       IF NOT #Positionen[20].Sperre AND NOT #Vorzug THEN
           "FC_FW_Auftrag_Befehl"(inQuelle := #tmpQuelle,
                                  inZiel := 20,
                                  Befehl_ok => #Befehl_ok,
                                  outQuelle => #Quelle,
                                  outZiel => #Ziel);

           #nextStep := NOT #Befehl_ok;
       ELSIF NOT #Positionen[24].Sperre THEN
           "FC_FW_Auftrag_Befehl"(inQuelle := #tmpQuelle,
                                  inZiel := 24,
                                  Befehl_ok => #Befehl_ok,
                                  outQuelle => #Quelle,
                                  outZiel => #Ziel);

           #nextStep := NOT #Befehl_ok;
       ELSE
           #nextStep := TRUE;
       END_IF;
       RETURN;
   END_IF;

   //
   #nextStep := TRUE;
END_REGION
END_FUNCTION

FUNCTION "FC_FW_Auftrag_Step1_NB" : Void   // FC181, LAD
TITLE = Schritt CM01/CMD02 -> CM03
{ S7_Optimized_Access := 'TRUE' }
// Ältesten Warenträger in CM01/CM02 suchen und nach CM03 transportieren
// stored: AutoNumber false, SetENOAutomatically false
   VAR_INPUT
      Frg_Schritt : Bool;
   END_VAR
   VAR_OUTPUT
      nextStep : Bool;
      startStep : Bool;
      parkStep : Bool;
   END_VAR
   VAR_IN_OUT
      Quelle : Int;
      Ziel : Int;
      Positionen : Array[1..30] of "UDT_Auftrag_Pos";
   END_VAR
   VAR_TEMP
      Sperre_Kurz_li : Bool;
      Sperre_Kurz_re : Bool;
      Sperre_Lang : Bool;
      Vorzug : Bool;
      Befehl_ok : Bool;
      tmpQuelle : Int;
      Oldest : Real;
   END_VAR
BEGIN

REGION Network 1 (SCL): Initialisieren
   IF (#Quelle <> 0) AND (#Ziel <> 0) THEN
       #nextStep := #Positionen[#Quelle].Sperre;
       #startStep := NOT #nextStep;
       #Quelle := 0;
       #Ziel := 0;
       RETURN;
   END_IF;

   #Quelle := 0;
   #Ziel := 0;
   #nextStep := FALSE;
   #startStep := FALSE;

   IF NOT #Frg_Schritt THEN
       #nextStep := TRUE;
       RETURN;
   END_IF;
END_REGION

REGION Network 2 (SCL): Positionen sperren
   //Groß links nicht möglich
   #Positionen[3].CheckSperre := #Positionen[9].Sperre;
   #Positionen[15].CheckSperre := #Positionen[9].Sperre;

   //Groß rechts nicht möglich
   #Positionen[4].CheckSperre := #Positionen[10].Sperre;
   #Positionen[16].CheckSperre := #Positionen[10].Sperre;

   //kein Platz für Kurz links in CM03
   #Sperre_Kurz_li := #Positionen[7].Sperre AND #Positionen[11].Sperre;

   //kein Platz für Kurz rechts in CM03
   #Sperre_Kurz_re := #Positionen[8].Sperre AND #Positionen[12].Sperre;

   //kein Platz für Lang in CM03
   #Sperre_Lang := (#Positionen[7].Sperre OR #Positionen[8].Sperre) AND (#Positionen[11].Sperre OR #Positionen[12].Sperre);

   //Lang in P1 oder
   //kein Platz auf rechter Seite
   //-> P2 sperren
   #Positionen[2].CheckSperre := #Sperre_Kurz_re OR (#Positionen[1].Wt_Typ = "WT_Typ_LS");

   //Lang in P1 und kein Platz für Lang oder
   //kein Platz auf linker Seite
   //-> P1 sperren
   #Positionen[1].CheckSperre := #Sperre_Kurz_li OR ((#Positionen[1].Wt_Typ = "WT_Typ_LS") AND #Sperre_Lang);

   //Lang in P5 oder
   //kein Platz auf rechter Seite
   //-> P6 sperren
   #Positionen[6].CheckSperre := #Sperre_Kurz_re OR (#Positionen[5].Wt_Typ = "WT_Typ_LS");

   //Lang in P5 und kein Platz für Lang oder
   //kein Platz auf linker Seite
   //-> P5 sperren
   #Positionen[5].CheckSperre := #Sperre_Kurz_li OR ((#Positionen[5].Wt_Typ = "WT_Typ_LS") AND #Sperre_Lang);

   //Lang in P13 oder
   //kein Platz auf rechter Seite
   //-> P14 sperren
   #Positionen[14].CheckSperre := #Sperre_Kurz_re OR (#Positionen[13].Wt_Typ = "WT_Typ_LS");

   //Lang in P13 und kein Platz für Lang oder
   //kein Platz auf linker Seite
   //-> P13 sperren
   #Positionen[13].CheckSperre := #Sperre_Kurz_li OR ((#Positionen[13].Wt_Typ = "WT_Typ_LS") AND #Sperre_Lang);

   //Lang in P17 oder
   //kein Platz auf rechter Seite
   //-> P18 sperren
   #Positionen[18].CheckSperre := #Sperre_Kurz_re OR (#Positionen[17].Wt_Typ = "WT_Typ_LS");

   //Lang in P17 und kein Platz für Lang oder
   //kein Platz auf linker Seite
   //-> P17 sperren
   #Positionen[17].CheckSperre := #Sperre_Kurz_li OR ((#Positionen[17].Wt_Typ = "WT_Typ_LS") AND #Sperre_Lang);
END_REGION

REGION Network 3 (SCL): Ältesten WT suchen
   //
   #Oldest := 0;
   #tmpQuelle := 0;

   //CM01
   "FC_FW_Auftrag_Suche"(Pos1 := 1,
                         Pos2 := 6,
                         Positionen := #Positionen,
                         Quelle := #tmpQuelle,
                         Oldest := #Oldest);

   //CM02
   "FC_FW_Auftrag_Suche"(Pos1 := 13,
                         Pos2 := 18,
                         Positionen := #Positionen,
                         Quelle := #tmpQuelle,
                         Oldest := #Oldest);
END_REGION

REGION Network 4 (SCL): Auswertung
   IF #tmpQuelle = 0 THEN
       //kein WT
       #nextStep := TRUE;
       RETURN;
   END_IF;

   IF ("DI_FW_1".ZST.POSITION_li <= 6) AND (#tmpQuelle <= 6) THEN
       //schieben wenn über Quelle CM01
       "FC_FW_Auftrag_Befehl"(inQuelle := 7,
                              inZiel := 0,
                              Befehl_ok => #Befehl_ok,
                              outQuelle => #Quelle,
                              outZiel => #Ziel);

       #nextStep := NOT #Befehl_ok;
       RETURN;
   END_IF;

   IF ("DI_FW_1".ZST.POSITION_li >= 13) AND ("DI_FW_1".ZST.POSITION_li <= 18) AND (#tmpQuelle >= 13) THEN
       //schieben wenn über Quelle CM02
       "FC_FW_Auftrag_Befehl"(inQuelle := 11,
                              inZiel := 0,
                              Befehl_ok => #Befehl_ok,
                              outQuelle => #Quelle,
                              outZiel => #Ziel);

       #nextStep := NOT #Befehl_ok;
       RETURN;
   END_IF;

   IF NOT #Positionen[#tmpQuelle].Fertig THEN
       #parkStep := TRUE;
       RETURN;
   END_IF;

   IF (#tmpQuelle = 3) OR (#tmpQuelle = 15) THEN
       //Gross links
       IF NOT #Positionen[9].Sperre THEN
           "FC_FW_Auftrag_Befehl"(inQuelle := #tmpQuelle,
                                  inZiel := 9,
                                  Befehl_ok => #Befehl_ok,
                                  outQuelle => #Quelle,
                                  outZiel => #Ziel);

           #nextStep := NOT #Befehl_ok;
       ELSE
           #nextStep := TRUE;
       END_IF;
       RETURN;
   END_IF;

   IF (#tmpQuelle = 4) OR (#tmpQuelle = 16) THEN
       //Gross rechts
       IF NOT #Positionen[10].Sperre THEN
           "FC_FW_Auftrag_Befehl"(inQuelle := #tmpQuelle,
                                  inZiel := 10,
                                  Befehl_ok => #Befehl_ok,
                                  outQuelle => #Quelle,
                                  outZiel => #Ziel);

           #nextStep := NOT #Befehl_ok;
       ELSE
           #nextStep := TRUE;
       END_IF;
       RETURN;
   END_IF;

   IF (#Positionen[#tmpQuelle].Wt_Typ = "WT_Typ_LS") AND ((#tmpQuelle = 1) OR (#tmpQuelle = 5) OR (#tmpQuelle = 13) OR (#tmpQuelle = 17)) THEN
       //Lang
       IF NOT #Positionen[7].Sperre AND NOT #Positionen[8].Sperre THEN
           "FC_FW_Auftrag_Befehl"(inQuelle := #tmpQuelle,
                                  inZiel := 7,
                                  Befehl_ok => #Befehl_ok,
                                  outQuelle => #Quelle,
                                  outZiel => #Ziel);

           #nextStep := NOT #Befehl_ok;
       ELSIF NOT #Positionen[11].Sperre AND NOT #Positionen[12].Sperre THEN
           "FC_FW_Auftrag_Befehl"(inQuelle := #tmpQuelle,
                                  inZiel := 11,
                                  Befehl_ok => #Befehl_ok,
                                  outQuelle => #Quelle,
                                  outZiel => #Ziel);

           #nextStep := NOT #Befehl_ok;
       ELSE
           #nextStep := TRUE;
       END_IF;
       RETURN;
   END_IF;

   IF (#tmpQuelle = 1) OR (#tmpQuelle = 5) OR (#tmpQuelle = 13) OR (#tmpQuelle = 17) THEN
       //Kurz links
       #Vorzug := NOT #Positionen[7].Sperre AND NOT #Positionen[8].Sperre AND NOT #Positionen[11].Sperre AND #Positionen[12].Sperre;

       IF NOT #Positionen[7].Sperre AND NOT #Vorzug THEN
           "FC_FW_Auftrag_Befehl"(inQuelle := #tmpQuelle,
                                  inZiel := 7,
                                  Befehl_ok => #Befehl_ok,
                                  outQuelle => #Quelle,
                                  outZiel => #Ziel);

           #nextStep := NOT #Befehl_ok;
       ELSIF NOT #Positionen[11].Sperre THEN
           "FC_FW_Auftrag_Befehl"(inQuelle := #tmpQuelle,
                                  inZiel := 11,
                                  Befehl_ok => #Befehl_ok,
                                  outQuelle => #Quelle,
                                  outZiel => #Ziel);

           #nextStep := NOT #Befehl_ok;
       ELSE
           #nextStep := TRUE;
       END_IF;
       RETURN;
   END_IF;

   IF (#tmpQuelle = 2) OR (#tmpQuelle = 6) OR (#tmpQuelle = 14) OR (#tmpQuelle = 18) THEN
       //Kurz rechts
       #Vorzug := NOT #Positionen[7].Sperre AND NOT #Positionen[8].Sperre AND #Positionen[11].Sperre AND NOT #Positionen[12].Sperre;

       IF NOT #Positionen[8].Sperre AND NOT #Vorzug THEN
           "FC_FW_Auftrag_Befehl"(inQuelle := #tmpQuelle,
                                  inZiel := 8,
                                  Befehl_ok => #Befehl_ok,
                                  outQuelle => #Quelle,
                                  outZiel => #Ziel);

           #nextStep := NOT #Befehl_ok;
       ELSIF NOT #Positionen[12].Sperre THEN
           "FC_FW_Auftrag_Befehl"(inQuelle := #tmpQuelle,
                                  inZiel := 12,
                                  Befehl_ok => #Befehl_ok,
                                  outQuelle => #Quelle,
                                  outZiel => #Ziel);

           #nextStep := NOT #Befehl_ok;
       ELSE
           #nextStep := TRUE;
       END_IF;
       RETURN;
   END_IF;

   //?
   #nextStep := TRUE;
END_REGION
END_FUNCTION

FUNCTION "FC_FW_Auftrag_Step2_KB" : Void   // FC1082, LAD
TITLE = Schritt CM03/CM04 -> CM01/CM02
{ S7_Optimized_Access := 'TRUE' }
// Ältesten Warenträger in CM03/CM04 suchen und nach CM01/CM02 transportieren
// stored: AutoNumber false, SetENOAutomatically false
   VAR_INPUT
      Frg_Schritt : Bool;
   END_VAR
   VAR_OUTPUT
      nextStep : Bool;
      startStep : Bool;
      parkStep : Bool;
   END_VAR
   VAR_IN_OUT
      Quelle : Int;
      Ziel : Int;
      Positionen : Array[1..30] of "UDT_Auftrag_Pos";
   END_VAR
   VAR_TEMP
      Sperre_Kurz_li_CM01 : Bool;
      Sperre_Kurz_re_CM01 : Bool;
      Sperre_Lang_CM01 : Bool;
      Sperre_Kurz_li_CM02 : Bool;
      Sperre_Kurz_re_CM02 : Bool;
      Sperre_Lang_CM02 : Bool;
      Vorzug : Bool;
      Vorzug1 : Bool;
      Vorzug2 : Bool;
      Befehl_ok : Bool;
      tmpQuelle : Int;
      Oldest : Real;
   END_VAR
   VAR CONSTANT
      Wt_Cmd_AetzenCM01 : Int := 1;
      Wt_Cmd_AetzenCM02 : Int := 13;
   END_VAR
BEGIN

REGION Network 1 (SCL)
   IF (#Quelle <> 0) AND (#Ziel <> 0) THEN
       #nextStep := #Positionen[#Quelle].Sperre;
       #startStep := NOT #nextStep;
       #Quelle := 0;
       #Ziel := 0;
       RETURN;
   END_IF;

   #Quelle := 0;
   #Ziel := 0;
   #nextStep := FALSE;
   #startStep := FALSE;

   IF NOT #Frg_Schritt THEN
       #nextStep := TRUE;
       RETURN;
   END_IF;
END_REGION

REGION Network 2 (SCL): Positionen sperren
   // GO nur "161"
   //Groß links nicht möglich
   #Positionen[9].CheckSperre := (#Positionen[3].Sperre ) OR (#Positionen[9].Wt_Cmd <> #Wt_Cmd_AetzenCM01);

   //Groß rechts nicht möglich
   #Positionen[10].CheckSperre := (#Positionen[4].Sperre AND #Positionen[16].Sperre) OR (#Positionen[10].Wt_Cmd <> #Wt_Cmd_AetzenCM01);

   //kein Platz für Kurz links in CM01
   #Sperre_Kurz_li_CM01 := #Positionen[1].Sperre AND #Positionen[5].Sperre;

   //kein Platz für Kurz links in CM02
   #Sperre_Kurz_li_CM02 := #Positionen[13].Sperre AND #Positionen[17].Sperre;

   //kein Platz für Kurz rechts in CM01
   #Sperre_Kurz_re_CM01 := #Positionen[2].Sperre AND #Positionen[6].Sperre;

   //kein Platz für Kurz rechts in CM02
   #Sperre_Kurz_re_CM02 := #Positionen[14].Sperre AND #Positionen[18].Sperre;

   //kein Platz für Lang in CM01
   #Sperre_Lang_CM01 := (#Positionen[1].Sperre OR #Positionen[2].Sperre) AND (#Positionen[5].Sperre OR #Positionen[6].Sperre);

   //kein Platz für Lang in CM02
   #Sperre_Lang_CM02:= (#Positionen[13].Sperre OR #Positionen[14].Sperre) AND (#Positionen[17].Sperre OR #Positionen[18].Sperre);

   //Lang in P7 oder
   //kein Platz auf rechter Seite
   //-> P8 sperren
   #Positionen[8].CheckSperre := #Sperre_Kurz_re_CM01 OR (#Positionen[7].Wt_Typ = "WT_Typ_LS") OR (#Positionen[8].Wt_Cmd <> #Wt_Cmd_AetzenCM01);

   //Lang in P7 und kein Platz für Lang oder
   //kein Platz auf linker Seite
   //-> P7 sperren
   #Positionen[7].CheckSperre := #Sperre_Kurz_li_CM01 OR ((#Positionen[7].Wt_Typ = "WT_Typ_LS") AND #Sperre_Lang_CM01) OR (#Positionen[7].Wt_Cmd <> #Wt_Cmd_AetzenCM01);

   //Lang in P7 oder
   //kein Platz auf rechter Seite
   //-> P12 sperren
   #Positionen[12].CheckSperre := #Sperre_Kurz_re_CM01 OR (#Positionen[11].Wt_Typ = "WT_Typ_LS") OR (#Positionen[12].Wt_Cmd <> #Wt_Cmd_AetzenCM01);

   //Lang in P11 und kein Platz für Lang oder
   //kein Platz auf linker Seite
   //-> P11 sperren
   #Positionen[11].CheckSperre := #Sperre_Kurz_li_CM01 OR ((#Positionen[11].Wt_Typ = "WT_Typ_LS") AND #Sperre_Lang_CM01) OR (#Positionen[11].Wt_Cmd <> #Wt_Cmd_AetzenCM01);

   //Lang in P19 oder
   //kein Platz auf rechter Seite
   //-> P20 sperren
   #Positionen[20].CheckSperre := #Sperre_Kurz_re_CM02 OR (#Positionen[19].Wt_Typ = "WT_Typ_LS") OR (#Positionen[20].Wt_Cmd <> #Wt_Cmd_AetzenCM02);

   //Lang in P19 und kein Platz für Lang oder
   //kein Platz auf linker Seite
   //-> P19 sperren
   #Positionen[19].CheckSperre := #Sperre_Kurz_li_CM02 OR ((#Positionen[19].Wt_Typ = "WT_Typ_LS") AND #Sperre_Lang_CM02) OR (#Positionen[19].Wt_Cmd <> #Wt_Cmd_AetzenCM02);

   //Lang in P23 oder
   //kein Platz auf rechter Seite
   //-> P24 sperren
   #Positionen[24].CheckSperre := #Sperre_Kurz_re_CM02 OR (#Positionen[23].Wt_Typ = "WT_Typ_LS") OR (#Positionen[24].Wt_Cmd <> #Wt_Cmd_AetzenCM02);

   //Lang in P23 und kein Platz für Lang oder
   //kein Platz auf linker Seite
   //-> P23 sperren
   #Positionen[23].CheckSperre := #Sperre_Kurz_li_CM02 OR ((#Positionen[23].Wt_Typ = "WT_Typ_LS") AND #Sperre_Lang_CM02) OR (#Positionen[23].Wt_Cmd <> #Wt_Cmd_AetzenCM02);
END_REGION

REGION Network 3 (SCL): Ältesten WT suchen
   //
   #Oldest := 0;
   #tmpQuelle := 0;

   //CM03
   "FC_FW_Auftrag_Suche"(Pos1 := 7,
                         Pos2 := 12,
                         Positionen := #Positionen,
                         Quelle := #tmpQuelle,
                         Oldest := #Oldest);

   //CM04
   "FC_FW_Auftrag_Suche"(Pos1 := 19,
                         Pos2 := 24,
                         Positionen := #Positionen,
                         Quelle := #tmpQuelle,
                         Oldest := #Oldest);
END_REGION

REGION Network 4 (SCL): Auswertung
   IF #tmpQuelle = 0 THEN
       //kein WT
       #nextStep := TRUE;
       RETURN;
   END_IF;

   IF NOT #Positionen[#tmpQuelle].Fertig THEN
       #parkStep := TRUE;
       RETURN;
   END_IF;

   IF (#tmpQuelle = 9) THEN
       //Gross links nur "161"
       IF NOT #Positionen[3].Sperre THEN
           "FC_FW_Auftrag_Befehl"(inQuelle := #tmpQuelle,
                                  inZiel := 3,
                                  Befehl_ok => #Befehl_ok,
                                  outQuelle => #Quelle,
                                  outZiel => #Ziel);

           #nextStep := NOT #Befehl_ok;
       ELSE
           #nextStep := TRUE;
       END_IF;
       RETURN;
   END_IF;

   IF (#tmpQuelle = 10) THEN
       //Gross rechts nur "161"
       IF NOT #Positionen[4].Sperre THEN
           "FC_FW_Auftrag_Befehl"(inQuelle := #tmpQuelle,
                                  inZiel := 4,
                                  Befehl_ok => #Befehl_ok,
                                  outQuelle => #Quelle,
                                  outZiel => #Ziel);

           #nextStep := NOT #Befehl_ok;
       ELSE
           #nextStep := TRUE;
       END_IF;
       RETURN;
   END_IF;

   IF (#Positionen[#tmpQuelle].Wt_Typ = "WT_Typ_LS") AND ((#tmpQuelle = 7) OR (#tmpQuelle = 11)) THEN
       //Lang "161"
       IF NOT #Positionen[5].Sperre AND NOT #Positionen[6].Sperre THEN
           "FC_FW_Auftrag_Befehl"(inQuelle := #tmpQuelle,
                                  inZiel := 5,
                                  Befehl_ok => #Befehl_ok,
                                  outQuelle => #Quelle,
                                  outZiel => #Ziel);

           #nextStep := NOT #Befehl_ok;
       ELSIF NOT #Positionen[1].Sperre AND NOT #Positionen[2].Sperre THEN
           "FC_FW_Auftrag_Befehl"(inQuelle := #tmpQuelle,
                                  inZiel := 1,
                                  Befehl_ok => #Befehl_ok,
                                  outQuelle => #Quelle,
                                  outZiel => #Ziel);

           #nextStep := NOT #Befehl_ok;
       ELSE
           #nextStep := TRUE;
       END_IF;
       RETURN;
   END_IF;

   IF (#Positionen[#tmpQuelle].Wt_Typ = "WT_Typ_LS") AND ((#tmpQuelle = 19) OR (#tmpQuelle = 23)) THEN
       //Lang "151"
       IF NOT #Positionen[17].Sperre AND NOT #Positionen[18].Sperre THEN
           "FC_FW_Auftrag_Befehl"(inQuelle := #tmpQuelle,
                                  inZiel := 17,
                                  Befehl_ok => #Befehl_ok,
                                  outQuelle => #Quelle,
                                  outZiel => #Ziel);

           #nextStep := NOT #Befehl_ok;
       ELSIF NOT #Positionen[13].Sperre AND NOT #Positionen[14].Sperre THEN
           "FC_FW_Auftrag_Befehl"(inQuelle := #tmpQuelle,
                                  inZiel := 13,
                                  Befehl_ok => #Befehl_ok,
                                  outQuelle => #Quelle,
                                  outZiel => #Ziel);

           #nextStep := NOT #Befehl_ok;
       ELSE
           #nextStep := TRUE;
       END_IF;
       RETURN;
   END_IF;

   IF (#tmpQuelle = 7) OR (#tmpQuelle = 11) THEN
       //Kurz links "161"
       #Vorzug1 := NOT #Positionen[1].Sperre AND #Positionen[2].Sperre;
       #Vorzug2 := NOT #Positionen[5].Sperre AND #Positionen[6].Sperre;

       #Vorzug := NOT #Vorzug2 AND #Vorzug1;
       IF NOT #Positionen[5].Sperre AND NOT #Vorzug THEN
           "FC_FW_Auftrag_Befehl"(inQuelle := #tmpQuelle,
                                  inZiel := 5,
                                  Befehl_ok => #Befehl_ok,
                                  outQuelle => #Quelle,
                                  outZiel => #Ziel);

           #nextStep := NOT #Befehl_ok;
           RETURN;
       END_IF;

       #Vorzug := NOT #Vorzug1 AND #Vorzug1;
       IF NOT #Positionen[1].Sperre AND NOT #Vorzug THEN
           "FC_FW_Auftrag_Befehl"(inQuelle := #tmpQuelle,
                                  inZiel := 1,
                                  Befehl_ok => #Befehl_ok,
                                  outQuelle => #Quelle,
                                  outZiel => #Ziel);

           #nextStep := NOT #Befehl_ok;
           RETURN;
       END_IF;

       #nextStep := TRUE;
       RETURN;
   END_IF;

   IF (#tmpQuelle = 8) OR (#tmpQuelle = 12) THEN
       //Kurz rechts "161"
       #Vorzug1 := NOT #Positionen[2].Sperre AND #Positionen[1].Sperre;
       #Vorzug2 := NOT #Positionen[6].Sperre AND #Positionen[5].Sperre;

       #Vorzug := NOT #Vorzug2 AND #Vorzug1;
       IF NOT #Positionen[6].Sperre AND NOT #Vorzug THEN
           "FC_FW_Auftrag_Befehl"(inQuelle := #tmpQuelle,
                                  inZiel := 6,
                                  Befehl_ok => #Befehl_ok,
                                  outQuelle => #Quelle,
                                  outZiel => #Ziel);

           #nextStep := NOT #Befehl_ok;
           RETURN;
       END_IF;


       #Vorzug := NOT #Vorzug1 AND #Vorzug2;
       IF NOT #Positionen[2].Sperre AND NOT #Vorzug THEN
           "FC_FW_Auftrag_Befehl"(inQuelle := #tmpQuelle,
                                  inZiel := 2,
                                  Befehl_ok => #Befehl_ok,
                                  outQuelle => #Quelle,
                                  outZiel => #Ziel);

           #nextStep := NOT #Befehl_ok;
           RETURN;
       END_IF;

       #nextStep := TRUE;
       RETURN;
   END_IF;

   IF (#tmpQuelle = 19) OR (#tmpQuelle = 23) THEN
       //Kurz links "151"
       #Vorzug1 := NOT #Positionen[13].Sperre AND #Positionen[14].Sperre;
       #Vorzug2 := NOT #Positionen[17].Sperre AND #Positionen[18].Sperre;

       #Vorzug := NOT #Vorzug2 AND #Vorzug1;
       IF NOT #Positionen[17].Sperre AND NOT #Vorzug THEN
           "FC_FW_Auftrag_Befehl"(inQuelle := #tmpQuelle,
                                  inZiel := 17,
                                  Befehl_ok => #Befehl_ok,
                                  outQuelle => #Quelle,
                                  outZiel => #Ziel);

           #nextStep := NOT #Befehl_ok;
           RETURN;
       END_IF;

       #Vorzug := NOT #Vorzug1 AND #Vorzug1;
       IF NOT #Positionen[13].Sperre AND NOT #Vorzug THEN
           "FC_FW_Auftrag_Befehl"(inQuelle := #tmpQuelle,
                                  inZiel := 13,
                                  Befehl_ok => #Befehl_ok,
                                  outQuelle => #Quelle,
                                  outZiel => #Ziel);

           #nextStep := NOT #Befehl_ok;
           RETURN;
       END_IF;

       #nextStep := TRUE;
       RETURN;
   END_IF;

   IF (#tmpQuelle = 20) OR (#tmpQuelle = 24) THEN
       //Kurz rechts "151"
       #Vorzug1 := NOT #Positionen[2].Sperre AND #Positionen[1].Sperre;
       #Vorzug2 := NOT #Positionen[6].Sperre AND #Positionen[5].Sperre;

       #Vorzug := NOT #Vorzug2 AND #Vorzug1;
       IF NOT #Positionen[18].Sperre AND NOT #Vorzug THEN
           "FC_FW_Auftrag_Befehl"(inQuelle := #tmpQuelle,
                                  inZiel := 18,
                                  Befehl_ok => #Befehl_ok,
                                  outQuelle => #Quelle,
                                  outZiel => #Ziel);

           #nextStep := NOT #Befehl_ok;
           RETURN;
       END_IF;

       #Vorzug := NOT #Vorzug1 AND #Vorzug2;
       IF NOT #Positionen[14].Sperre AND NOT #Vorzug THEN
           "FC_FW_Auftrag_Befehl"(inQuelle := #tmpQuelle,
                                  inZiel := 14,
                                  Befehl_ok => #Befehl_ok,
                                  outQuelle => #Quelle,
                                  outZiel => #Ziel);

           #nextStep := NOT #Befehl_ok;
           RETURN;
       END_IF;

       #nextStep := TRUE;
       RETURN;
   END_IF;

   //
   #nextStep := TRUE;
END_REGION
END_FUNCTION

FUNCTION "FC_FW_Auftrag_Step2_NB" : Void   // FC182, LAD
TITLE = Schritt CM03 -> CM01/CM02
{ S7_Optimized_Access := 'TRUE' }
// Ältesten Warenträger in CM03 suchen und nach CM01/CM02 transportieren
// stored: AutoNumber false, SetENOAutomatically false
   VAR_INPUT
      Frg_Schritt : Bool;
   END_VAR
   VAR_OUTPUT
      nextStep : Bool;
      startStep : Bool;
      parkStep : Bool;
   END_VAR
   VAR_IN_OUT
      Quelle : Int;
      Ziel : Int;
      Positionen : Array[1..30] of "UDT_Auftrag_Pos";
   END_VAR
   VAR_TEMP
      Sperre_Kurz_li : Bool;
      Sperre_Kurz_re : Bool;
      Sperre_Lang : Bool;
      Vorzug : Bool;
      Vorzug1 : Bool;
      Vorzug2 : Bool;
      Vorzug3 : Bool;
      Vorzug4 : Bool;
      Befehl_ok : Bool;
      tmpQuelle : Int;
      Oldest : Real;
   END_VAR
   VAR CONSTANT
      Wt_Cmd_Aetzen : Int := 1;
   END_VAR
BEGIN

REGION Network 1 (SCL)
   IF (#Quelle <> 0) AND (#Ziel <> 0) THEN
       #nextStep := #Positionen[#Quelle].Sperre;
       #startStep := NOT #nextStep;
       #Quelle := 0;
       #Ziel := 0;
       RETURN;
   END_IF;

   #Quelle := 0;
   #Ziel := 0;
   #nextStep := FALSE;
   #startStep := FALSE;

   IF NOT #Frg_Schritt THEN
       #nextStep := TRUE;
       RETURN;
   END_IF;
END_REGION

REGION Network 2 (SCL): Positionen sperren
   //Groß links nicht möglich
   #Positionen[9].CheckSperre := (#Positionen[3].Sperre AND #Positionen[15].Sperre) OR (#Positionen[9].Wt_Cmd <> #Wt_Cmd_Aetzen);

   //Groß rechts nicht möglich
   #Positionen[10].CheckSperre := (#Positionen[4].Sperre AND #Positionen[16].Sperre) OR (#Positionen[10].Wt_Cmd <> #Wt_Cmd_Aetzen);

   //kein Platz für Kurz links in CM01/CM02
   #Sperre_Kurz_li := #Positionen[1].Sperre AND #Positionen[5].Sperre AND #Positionen[13].Sperre AND #Positionen[17].Sperre;

   //kein Platz für Kurz rechts in CM01/CM02
   #Sperre_Kurz_re := #Positionen[2].Sperre AND #Positionen[6].Sperre AND #Positionen[14].Sperre AND #Positionen[18].Sperre;

   //kein Platz für Lang in CM01/CM02
   #Sperre_Lang := (#Positionen[1].Sperre OR #Positionen[2].Sperre) AND (#Positionen[5].Sperre OR #Positionen[6].Sperre) AND (#Positionen[13].Sperre OR #Positionen[14].Sperre) AND (#Positionen[17].Sperre OR #Positionen[18].Sperre);

   //Lang in P7 oder
   //kein Platz auf rechter Seite
   //-> P8 sperren
   #Positionen[8].CheckSperre := #Sperre_Kurz_re OR (#Positionen[7].Wt_Typ = "WT_Typ_LS") OR (#Positionen[8].Wt_Cmd <> #Wt_Cmd_Aetzen);

   //Lang in P7 und kein Platz für Lang oder
   //kein Platz auf linker Seite
   //-> P7 sperren
   #Positionen[7].CheckSperre := #Sperre_Kurz_li OR ((#Positionen[7].Wt_Typ = "WT_Typ_LS") AND #Sperre_Lang) OR (#Positionen[7].Wt_Cmd <> #Wt_Cmd_Aetzen);

   //Lang in P11 oder
   //kein Platz auf rechter Seite
   //-> P12 sperren
   #Positionen[12].CheckSperre := #Sperre_Kurz_re OR (#Positionen[11].Wt_Typ = "WT_Typ_LS") OR (#Positionen[12].Wt_Cmd <> #Wt_Cmd_Aetzen);

   //Lang in P11 und kein Platz für Lang oder
   //kein Platz auf linker Seite
   //-> P11 sperren
   #Positionen[11].CheckSperre := #Sperre_Kurz_li OR ((#Positionen[11].Wt_Typ = "WT_Typ_LS") AND #Sperre_Lang) OR (#Positionen[11].Wt_Cmd <> #Wt_Cmd_Aetzen);
END_REGION

REGION Network 3 (SCL): Ältesten WT suchen
   //
   #Oldest := 0;
   #tmpQuelle := 0;

   //CM03
   "FC_FW_Auftrag_Suche"(Pos1 := 7,
                         Pos2 := 12,
                         Positionen := #Positionen,
                         Quelle := #tmpQuelle,
                         Oldest := #Oldest);
END_REGION

REGION Network 4 (SCL): Auswertung
   IF #tmpQuelle = 0 THEN
       //kein WT
       #nextStep := TRUE;
       RETURN;
   END_IF;

   IF NOT #Positionen[#tmpQuelle].Fertig THEN
       #parkStep := TRUE;
       RETURN;
   END_IF;

   IF (#tmpQuelle = 9) THEN
       //Gross links
       IF NOT #Positionen[3].Sperre THEN
           "FC_FW_Auftrag_Befehl"(inQuelle := #tmpQuelle,
                                  inZiel := 3,
                                  Befehl_ok => #Befehl_ok,
                                  outQuelle => #Quelle,
                                  outZiel => #Ziel);

           #nextStep := NOT #Befehl_ok;
       ELSIF NOT #Positionen[15].Sperre THEN
           "FC_FW_Auftrag_Befehl"(inQuelle := #tmpQuelle,
                                  inZiel := 15,
                                  Befehl_ok => #Befehl_ok,
                                  outQuelle => #Quelle,
                                  outZiel => #Ziel);

           #nextStep := NOT #Befehl_ok;
       ELSE
           #nextStep := TRUE;
       END_IF;
       RETURN;
   END_IF;

   IF (#tmpQuelle = 10) THEN
       //Gross rechts
       IF NOT #Positionen[4].Sperre THEN
           "FC_FW_Auftrag_Befehl"(inQuelle := #tmpQuelle,
                                  inZiel := 4,
                                  Befehl_ok => #Befehl_ok,
                                  outQuelle => #Quelle,
                                  outZiel => #Ziel);

           #nextStep := NOT #Befehl_ok;
       ELSIF NOT #Positionen[16].Sperre THEN
           "FC_FW_Auftrag_Befehl"(inQuelle := #tmpQuelle,
                                  inZiel := 16,
                                  Befehl_ok => #Befehl_ok,
                                  outQuelle => #Quelle,
                                  outZiel => #Ziel);

           #nextStep := NOT #Befehl_ok;
       ELSE
           #nextStep := TRUE;
       END_IF;
       RETURN;
   END_IF;

   IF (#Positionen[#tmpQuelle].Wt_Typ = "WT_Typ_LS") AND ((#tmpQuelle = 7) OR (#tmpQuelle = 11)) THEN
       //Lang
       IF NOT #Positionen[13].Sperre AND NOT #Positionen[14].Sperre THEN
           "FC_FW_Auftrag_Befehl"(inQuelle := #tmpQuelle,
                                  inZiel := 13,
                                  Befehl_ok => #Befehl_ok,
                                  outQuelle => #Quelle,
                                  outZiel => #Ziel);

           #nextStep := NOT #Befehl_ok;
       ELSIF NOT #Positionen[5].Sperre AND NOT #Positionen[6].Sperre THEN
           "FC_FW_Auftrag_Befehl"(inQuelle := #tmpQuelle,
                                  inZiel := 5,
                                  Befehl_ok => #Befehl_ok,
                                  outQuelle => #Quelle,
                                  outZiel => #Ziel);

           #nextStep := NOT #Befehl_ok;
       ELSIF NOT #Positionen[1].Sperre AND NOT #Positionen[2].Sperre THEN
           "FC_FW_Auftrag_Befehl"(inQuelle := #tmpQuelle,
                                  inZiel := 1,
                                  Befehl_ok => #Befehl_ok,
                                  outQuelle => #Quelle,
                                  outZiel => #Ziel);

           #nextStep := NOT #Befehl_ok;
       ELSIF NOT #Positionen[17].Sperre AND NOT #Positionen[18].Sperre THEN
           "FC_FW_Auftrag_Befehl"(inQuelle := #tmpQuelle,
                                  inZiel := 17,
                                  Befehl_ok => #Befehl_ok,
                                  outQuelle => #Quelle,
                                  outZiel => #Ziel);

           #nextStep := NOT #Befehl_ok;
       ELSE
           #nextStep := TRUE;
       END_IF;
       RETURN;
   END_IF;

   IF (#tmpQuelle = 7) OR (#tmpQuelle = 11) THEN
       //Kurz links
       #Vorzug1 := NOT #Positionen[1].Sperre AND #Positionen[2].Sperre;
       #Vorzug2 := NOT #Positionen[5].Sperre AND #Positionen[6].Sperre;
       #Vorzug3 := NOT #Positionen[13].Sperre AND #Positionen[14].Sperre;
       #Vorzug4 := NOT #Positionen[17].Sperre AND #Positionen[18].Sperre;

       #Vorzug := NOT #Vorzug2 AND (#Vorzug1 OR #Vorzug3 OR #Vorzug4);
       IF NOT #Positionen[5].Sperre AND NOT #Vorzug THEN
           "FC_FW_Auftrag_Befehl"(inQuelle := #tmpQuelle,
                                  inZiel := 5,
                                  Befehl_ok => #Befehl_ok,
                                  outQuelle => #Quelle,
                                  outZiel => #Ziel);

           #nextStep := NOT #Befehl_ok;
           RETURN;
       END_IF;

       #Vorzug := NOT #Vorzug3 AND (#Vorzug1 OR #Vorzug4);
       IF NOT #Positionen[13].Sperre AND NOT #Vorzug THEN
           "FC_FW_Auftrag_Befehl"(inQuelle := #tmpQuelle,
                                  inZiel := 13,
                                  Befehl_ok => #Befehl_ok,
                                  outQuelle => #Quelle,
                                  outZiel => #Ziel);

           #nextStep := NOT #Befehl_ok;
           RETURN;
       END_IF;

       #Vorzug := NOT #Vorzug1 AND #Vorzug4;
       IF NOT #Positionen[1].Sperre AND NOT #Vorzug THEN
           "FC_FW_Auftrag_Befehl"(inQuelle := #tmpQuelle,
                                  inZiel := 1,
                                  Befehl_ok => #Befehl_ok,
                                  outQuelle => #Quelle,
                                  outZiel => #Ziel);

           #nextStep := NOT #Befehl_ok;
           RETURN;
       END_IF;

       IF NOT #Positionen[17].Sperre THEN
           "FC_FW_Auftrag_Befehl"(inQuelle := #tmpQuelle,
                                  inZiel := 17,
                                  Befehl_ok => #Befehl_ok,
                                  outQuelle => #Quelle,
                                  outZiel => #Ziel);

           #nextStep := NOT #Befehl_ok;
           RETURN;
       END_IF;

       #nextStep := TRUE;
       RETURN;
   END_IF;

   IF (#tmpQuelle = 8) OR (#tmpQuelle = 12) THEN
       //Kurz rechts
       #Vorzug1 := NOT #Positionen[2].Sperre AND #Positionen[1].Sperre;
       #Vorzug2 := NOT #Positionen[6].Sperre AND #Positionen[5].Sperre;
       #Vorzug3 := NOT #Positionen[14].Sperre AND #Positionen[13].Sperre;
       #Vorzug4 := NOT #Positionen[18].Sperre AND #Positionen[17].Sperre;

       #Vorzug := NOT #Vorzug2 AND (#Vorzug1 OR #Vorzug3 OR #Vorzug4);
       IF NOT #Positionen[6].Sperre AND NOT #Vorzug THEN
           "FC_FW_Auftrag_Befehl"(inQuelle := #tmpQuelle,
                                  inZiel := 6,
                                  Befehl_ok => #Befehl_ok,
                                  outQuelle => #Quelle,
                                  outZiel => #Ziel);

           #nextStep := NOT #Befehl_ok;
           RETURN;
       END_IF;

       #Vorzug := NOT #Vorzug3 AND (#Vorzug1 OR #Vorzug4);
       IF NOT #Positionen[14].Sperre AND NOT #Vorzug THEN
           "FC_FW_Auftrag_Befehl"(inQuelle := #tmpQuelle,
                                  inZiel := 14,
                                  Befehl_ok => #Befehl_ok,
                                  outQuelle => #Quelle,
                                  outZiel => #Ziel);

           #nextStep := NOT #Befehl_ok;
           RETURN;
       END_IF;

       #Vorzug := NOT #Vorzug1 AND #Vorzug4;
       IF NOT #Positionen[2].Sperre AND NOT #Vorzug THEN
           "FC_FW_Auftrag_Befehl"(inQuelle := #tmpQuelle,
                                  inZiel := 2,
                                  Befehl_ok => #Befehl_ok,
                                  outQuelle => #Quelle,
                                  outZiel => #Ziel);

           #nextStep := NOT #Befehl_ok;
           RETURN;
       END_IF;

       IF NOT #Positionen[18].Sperre THEN
           "FC_FW_Auftrag_Befehl"(inQuelle := #tmpQuelle,
                                  inZiel := 18,
                                  Befehl_ok => #Befehl_ok,
                                  outQuelle => #Quelle,
                                  outZiel => #Ziel);

           #nextStep := NOT #Befehl_ok;
           RETURN;
       END_IF;

       #nextStep := TRUE;
       RETURN;
   END_IF;

   //?
   #nextStep := TRUE;
END_REGION
END_FUNCTION

FUNCTION "FC_FW_Auftrag_Step3_KB" : Void   // FC1083, LAD
TITLE = Schritt CM03 -> CM03 CM04-> CM04
{ S7_Optimized_Access := 'TRUE' }
// Ältesten Warenträger in CM03 / CM04 suchen und wieder einsetzen
// stored: AutoNumber false, SetENOAutomatically false
   VAR_INPUT
      Frg_Schritt : Bool;
   END_VAR
   VAR_OUTPUT
      nextStep : Bool;
      startStep : Bool;
      parkStep : Bool;
   END_VAR
   VAR_IN_OUT
      Quelle : Int;
      Ziel : Int;
      Positionen : Array[1..30] of "UDT_Auftrag_Pos";
   END_VAR
   VAR_TEMP
      Sperre_Kurz_li : Bool;
      Sperre_Kurz_re : Bool;
      Sperre_Lang : Bool;
      Vorzug : Bool;
      Befehl_ok : Bool;
      tmpQuelle : Int;
      Oldest : Real;
   END_VAR
   VAR CONSTANT
      Wt_Cmd_Spuele_CM03 : Int := 7;
      Wt_Cmd_Spuele_CM04 : Int := 19;
   END_VAR
BEGIN

REGION Network 1 (SCL)
   IF (#Quelle <> 0) AND (#Ziel <> 0) THEN
       #nextStep := #Positionen[#Quelle].Sperre;
       #startStep := NOT #nextStep;
       #Quelle := 0;
       #Ziel := 0;
       RETURN;
   END_IF;

   #Quelle := 0;
   #Ziel := 0;
   #nextStep := FALSE;
   #startStep := FALSE;

   IF NOT #Frg_Schritt THEN
       #nextStep := TRUE;
       RETURN;
   END_IF;
END_REGION

REGION Network 2 (SCL): Positionen sperren
   //Groß links nicht möglich
   #Positionen[9].CheckSperre := #Positionen[9].Wt_Cmd <> #Wt_Cmd_Spuele_CM03;

   //Groß rechts nicht möglich
   #Positionen[10].CheckSperre := #Positionen[10].Wt_Cmd <> #Wt_Cmd_Spuele_CM03;

   //Platz spielt keine Rolle, nur CMD

   //Lang in P7
   //-> P8 sperren
   #Positionen[8].CheckSperre := (#Positionen[7].Wt_Typ = "WT_Typ_LS") OR (#Positionen[8].Wt_Cmd <> #Wt_Cmd_Spuele_CM03);

   //-> P7 sperren
   #Positionen[7].CheckSperre := (#Positionen[7].Wt_Cmd <> #Wt_Cmd_Spuele_CM03);

   //Lang in P11 
   //-> P12 sperren
   #Positionen[12].CheckSperre := (#Positionen[11].Wt_Typ = "WT_Typ_LS") OR (#Positionen[12].Wt_Cmd <> #Wt_Cmd_Spuele_CM03);

   //Lang in P11
   //-> P11 sperren
   #Positionen[11].CheckSperre := (#Positionen[11].Wt_Cmd <> #Wt_Cmd_Spuele_CM03);

   //Lang in P19
   //-> P20 sperren
   #Positionen[20].CheckSperre := (#Positionen[19].Wt_Typ = "WT_Typ_LS") OR (#Positionen[20].Wt_Cmd <> #Wt_Cmd_Spuele_CM04);

   //-> P19 sperren
   #Positionen[19].CheckSperre := (#Positionen[19].Wt_Cmd <> #Wt_Cmd_Spuele_CM04);

   //Lang in P23 
   //-> P24 sperren
   #Positionen[24].CheckSperre := (#Positionen[23].Wt_Typ = "WT_Typ_LS") OR (#Positionen[24].Wt_Cmd = #Wt_Cmd_Spuele_CM04);

   //Lang in P23
   //-> P23 sperren
   #Positionen[23].CheckSperre := (#Positionen[23].Wt_Cmd <> #Wt_Cmd_Spuele_CM04);
END_REGION

REGION Network 3 (SCL): Ältesten WT suchen
   //
   #Oldest := 0;
   #tmpQuelle := 0;

   //CM03
   "FC_FW_Auftrag_Suche"(Pos1 := 7,
                         Pos2 := 12,
                         Positionen := #Positionen,
                         Quelle := #tmpQuelle,
                         Oldest := #Oldest);

   //CM04
   "FC_FW_Auftrag_Suche"(Pos1 := 19,
                         Pos2 := 24,
                         Positionen := #Positionen,
                         Quelle := #tmpQuelle,
                         Oldest := #Oldest);
END_REGION

REGION Network 4 (SCL): Auswertung
   IF #tmpQuelle = 0 THEN
       //kein WT
       #nextStep := TRUE;
       RETURN;
   END_IF;

   IF NOT #Positionen[#tmpQuelle].Fertig THEN
       #parkStep := TRUE;
       RETURN;
   END_IF;

   IF (#tmpQuelle = 9) THEN
       //Gross links - nur 161

           "FC_FW_Auftrag_Befehl"(inQuelle := #tmpQuelle,
                                  inZiel := 9,
                                  Befehl_ok => #Befehl_ok,
                                  outQuelle => #Quelle,
                                  outZiel => #Ziel);

           #nextStep := NOT #Befehl_ok;

       RETURN;
   END_IF;

   IF (#tmpQuelle = 10) THEN
       //Gross rechts - nur "161"

           "FC_FW_Auftrag_Befehl"(inQuelle := #tmpQuelle,
                                  inZiel := 10,
                                  Befehl_ok => #Befehl_ok,
                                  outQuelle => #Quelle,
                                  outZiel => #Ziel);

           #nextStep := NOT #Befehl_ok;

       RETURN;
   END_IF;

   IF (#Positionen[#tmpQuelle].Wt_Typ = "WT_Typ_LS") AND (#tmpQuelle = 7) THEN
       //Lang "161"
       "FC_FW_Auftrag_Befehl"(inQuelle := #tmpQuelle,
                                  inZiel := 7,
                                  Befehl_ok => #Befehl_ok,
                                  outQuelle => #Quelle,
                                  outZiel => #Ziel);

           #nextStep := NOT #Befehl_ok;

        RETURN;
   END_IF;


   IF (#Positionen[#tmpQuelle].Wt_Typ = "WT_Typ_LS") AND (#tmpQuelle = 11) THEN
       //Lang "161"
       "FC_FW_Auftrag_Befehl"(inQuelle := #tmpQuelle,
                              inZiel := 11,
                              Befehl_ok => #Befehl_ok,
                              outQuelle => #Quelle,
                              outZiel => #Ziel);

       #nextStep := NOT #Befehl_ok;

       RETURN;
   END_IF;

   IF (#Positionen[#tmpQuelle].Wt_Typ = "WT_Typ_LS") AND (#tmpQuelle = 19) THEN
       //Lang "151"
       "FC_FW_Auftrag_Befehl"(inQuelle := #tmpQuelle,
                              inZiel := 19,
                              Befehl_ok => #Befehl_ok,
                              outQuelle => #Quelle,
                              outZiel => #Ziel);

       #nextStep := NOT #Befehl_ok;

       RETURN;
   END_IF;


   IF (#Positionen[#tmpQuelle].Wt_Typ = "WT_Typ_LS") AND (#tmpQuelle = 23) THEN
       //Lang "151"
       "FC_FW_Auftrag_Befehl"(inQuelle := #tmpQuelle,
                              inZiel := 23,
                              Befehl_ok => #Befehl_ok,
                              outQuelle => #Quelle,
                              outZiel => #Ziel);

       #nextStep := NOT #Befehl_ok;

       RETURN;
   END_IF;


   IF (#tmpQuelle = 7) THEN
       //Kurz links "161
       "FC_FW_Auftrag_Befehl"(inQuelle := #tmpQuelle,
                                  inZiel := 7,
                                  Befehl_ok => #Befehl_ok,
                                  outQuelle => #Quelle,
                                  outZiel => #Ziel);

           #nextStep := NOT #Befehl_ok;
           RETURN;
   END_IF;

   IF (#tmpQuelle = 11) THEN
       //Kurz links "161
       "FC_FW_Auftrag_Befehl"(inQuelle := #tmpQuelle,
                              inZiel := 11,
                              Befehl_ok => #Befehl_ok,
                              outQuelle => #Quelle,
                              outZiel => #Ziel);

       #nextStep := NOT #Befehl_ok;
       RETURN;
   END_IF;

   IF (#tmpQuelle = 8) THEN
       //Kurz rechtss "161
       "FC_FW_Auftrag_Befehl"(inQuelle := #tmpQuelle,
                              inZiel := 8,
                              Befehl_ok => #Befehl_ok,
                              outQuelle => #Quelle,
                              outZiel => #Ziel);

       #nextStep := NOT #Befehl_ok;
       RETURN;
   END_IF;

   IF (#tmpQuelle = 12) THEN
       //Kurz rechts "161
       "FC_FW_Auftrag_Befehl"(inQuelle := #tmpQuelle,
                              inZiel := 12,
                              Befehl_ok => #Befehl_ok,
                              outQuelle => #Quelle,
                              outZiel => #Ziel);

       #nextStep := NOT #Befehl_ok;
       RETURN;
   END_IF;


   IF (#tmpQuelle = 19) THEN
       //Kurz links "151
       "FC_FW_Auftrag_Befehl"(inQuelle := #tmpQuelle,
                              inZiel := 19,
                              Befehl_ok => #Befehl_ok,
                              outQuelle => #Quelle,
                              outZiel => #Ziel);

       #nextStep := NOT #Befehl_ok;
       RETURN;
   END_IF;

   IF (#tmpQuelle = 23) THEN
       //Kurz links "151
       "FC_FW_Auftrag_Befehl"(inQuelle := #tmpQuelle,
                              inZiel := 23,
                              Befehl_ok => #Befehl_ok,
                              outQuelle => #Quelle,
                              outZiel => #Ziel);

       #nextStep := NOT #Befehl_ok;
       RETURN;
   END_IF;

   IF (#tmpQuelle = 20) THEN
       //Kurz rechtss "151
       "FC_FW_Auftrag_Befehl"(inQuelle := #tmpQuelle,
                              inZiel := 20,
                              Befehl_ok => #Befehl_ok,
                              outQuelle => #Quelle,
                              outZiel => #Ziel);

       #nextStep := NOT #Befehl_ok;
       RETURN;
   END_IF;

   IF (#tmpQuelle = 24) THEN
       //Kurz rechts "151
       "FC_FW_Auftrag_Befehl"(inQuelle := #tmpQuelle,
                              inZiel := 24,
                              Befehl_ok => #Befehl_ok,
                              outQuelle => #Quelle,
                              outZiel => #Ziel);

       #nextStep := NOT #Befehl_ok;
       RETURN;
   END_IF;
   //
   #nextStep := TRUE;
END_REGION
END_FUNCTION

FUNCTION "FC_FW_Auftrag_Step3_NB" : Void   // FC183, LAD
TITLE = Schritt CM03 -> CM04
{ S7_Optimized_Access := 'TRUE' }
// Ältesten Warenträger in CM03 suchen und nach CM04 transportieren
// stored: AutoNumber false, SetENOAutomatically false
   VAR_INPUT
      Frg_Schritt : Bool;
   END_VAR
   VAR_OUTPUT
      nextStep : Bool;
      startStep : Bool;
      parkStep : Bool;
   END_VAR
   VAR_IN_OUT
      Quelle : Int;
      Ziel : Int;
      Positionen : Array[1..30] of "UDT_Auftrag_Pos";
   END_VAR
   VAR_TEMP
      Sperre_Kurz_li : Bool;
      Sperre_Kurz_re : Bool;
      Sperre_Lang : Bool;
      Vorzug : Bool;
      Befehl_ok : Bool;
      tmpQuelle : Int;
      Oldest : Real;
   END_VAR
   VAR CONSTANT
      Wt_Cmd_Aetzen : Int := 1;
   END_VAR
BEGIN

REGION Network 1 (SCL)
   IF (#Quelle <> 0) AND (#Ziel <> 0) THEN
       #nextStep := #Positionen[#Quelle].Sperre;
       #startStep := NOT #nextStep;
       #Quelle := 0;
       #Ziel := 0;
       RETURN;
   END_IF;

   #Quelle := 0;
   #Ziel := 0;
   #nextStep := FALSE;
   #startStep := FALSE;

   IF NOT #Frg_Schritt THEN
       #nextStep := TRUE;
       RETURN;
   END_IF;
END_REGION

REGION Network 2 (SCL): Positionen sperren
   //Groß links nicht möglich
   #Positionen[9].CheckSperre := #Positionen[21].Sperre OR (#Positionen[9].Wt_Cmd = #Wt_Cmd_Aetzen);

   //Groß rechts nicht möglich
   #Positionen[10].CheckSperre := #Positionen[22].Sperre OR (#Positionen[10].Wt_Cmd = #Wt_Cmd_Aetzen);

   //kein Platz für Kurz links in CM04
   #Sperre_Kurz_li := #Positionen[19].Sperre AND #Positionen[23].Sperre;

   //kein Platz für Kurz rechts in CM04
   #Sperre_Kurz_re := #Positionen[20].Sperre AND #Positionen[24].Sperre;

   //kein Platz für Lang in CM04
   #Sperre_Lang := (#Positionen[19].Sperre OR #Positionen[20].Sperre) AND (#Positionen[23].Sperre OR #Positionen[24].Sperre);

   //Lang in P7 oder
   //kein Platz auf rechter Seite
   //-> P8 sperren
   #Positionen[8].CheckSperre := #Sperre_Kurz_re OR (#Positionen[7].Wt_Typ = "WT_Typ_LS") OR (#Positionen[8].Wt_Cmd = #Wt_Cmd_Aetzen);

   //Lang in P7 und kein Platz für Lang oder
   //kein Platz auf linker Seite
   //-> P7 sperren
   #Positionen[7].CheckSperre := #Sperre_Kurz_li OR ((#Positionen[7].Wt_Typ = "WT_Typ_LS") AND #Sperre_Lang) OR (#Positionen[7].Wt_Cmd = #Wt_Cmd_Aetzen);

   //Lang in P11 oder
   //kein Platz auf rechter Seite
   //-> P12 sperren
   #Positionen[12].CheckSperre := #Sperre_Kurz_re OR (#Positionen[11].Wt_Typ = "WT_Typ_LS") OR (#Positionen[12].Wt_Cmd = #Wt_Cmd_Aetzen);

   //Lang in P11 und kein Platz für Lang oder
   //kein Platz auf linker Seite
   //-> P11 sperren
   #Positionen[11].CheckSperre := #Sperre_Kurz_li OR ((#Positionen[11].Wt_Typ = "WT_Typ_LS") AND #Sperre_Lang) OR (#Positionen[11].Wt_Cmd = #Wt_Cmd_Aetzen);
END_REGION

REGION Network 3 (SCL): Ältesten WT suchen
   //
   #Oldest := 0;
   #tmpQuelle := 0;

   //CM03
   "FC_FW_Auftrag_Suche"(Pos1 := 7,
                         Pos2 := 12,
                         Positionen := #Positionen,
                         Quelle := #tmpQuelle,
                         Oldest := #Oldest);
END_REGION

REGION Network 4 (SCL): Auswertung
   IF #tmpQuelle = 0 THEN
       //kein WT
       #nextStep := TRUE;
       RETURN;
   END_IF;

   IF NOT #Positionen[#tmpQuelle].Fertig THEN
       #parkStep := TRUE;
       RETURN;
   END_IF;

   IF (#tmpQuelle = 9) THEN
       //Gross links
       IF NOT #Positionen[21].Sperre THEN
           "FC_FW_Auftrag_Befehl"(inQuelle := #tmpQuelle,
                                  inZiel := 21,
                                  Befehl_ok => #Befehl_ok,
                                  outQuelle => #Quelle,
                                  outZiel => #Ziel);

           #nextStep := NOT #Befehl_ok;
       ELSE
           #nextStep := TRUE;
       END_IF;
       RETURN;
   END_IF;

   IF (#tmpQuelle = 10) THEN
       //Gross rechts
       IF NOT #Positionen[22].Sperre THEN
           "FC_FW_Auftrag_Befehl"(inQuelle := #tmpQuelle,
                                  inZiel := 22,
                                  Befehl_ok => #Befehl_ok,
                                  outQuelle => #Quelle,
                                  outZiel => #Ziel);

           #nextStep := NOT #Befehl_ok;
       ELSE
           #nextStep := TRUE;
       END_IF;
       RETURN;
   END_IF;

   IF (#Positionen[#tmpQuelle].Wt_Typ = "WT_Typ_LS") AND ((#tmpQuelle = 7) OR (#tmpQuelle = 11)) THEN
       //Lang
       IF NOT #Positionen[19].Sperre AND NOT #Positionen[20].Sperre THEN
           "FC_FW_Auftrag_Befehl"(inQuelle := #tmpQuelle,
                                  inZiel := 19,
                                  Befehl_ok => #Befehl_ok,
                                  outQuelle => #Quelle,
                                  outZiel => #Ziel);

           #nextStep := NOT #Befehl_ok;
       ELSIF NOT #Positionen[23].Sperre AND NOT #Positionen[24].Sperre THEN
           "FC_FW_Auftrag_Befehl"(inQuelle := #tmpQuelle,
                                  inZiel := 23,
                                  Befehl_ok => #Befehl_ok,
                                  outQuelle => #Quelle,
                                  outZiel => #Ziel);

           #nextStep := NOT #Befehl_ok;
       ELSE
           #nextStep := TRUE;
       END_IF;
       RETURN;
   END_IF;

   IF (#tmpQuelle = 7) OR (#tmpQuelle = 11) THEN
       //Kurz links
       #Vorzug := NOT #Positionen[19].Sperre AND NOT #Positionen[20].Sperre AND NOT #Positionen[23].Sperre AND #Positionen[24].Sperre;

       IF NOT #Positionen[19].Sperre AND NOT #Vorzug THEN
           "FC_FW_Auftrag_Befehl"(inQuelle := #tmpQuelle,
                                  inZiel := 19,
                                  Befehl_ok => #Befehl_ok,
                                  outQuelle => #Quelle,
                                  outZiel => #Ziel);

           #nextStep := NOT #Befehl_ok;
       ELSIF NOT #Positionen[23].Sperre THEN
           "FC_FW_Auftrag_Befehl"(inQuelle := #tmpQuelle,
                                  inZiel := 23,
                                  Befehl_ok => #Befehl_ok,
                                  outQuelle => #Quelle,
                                  outZiel => #Ziel);

           #nextStep := NOT #Befehl_ok;
       ELSE
           #nextStep := TRUE;
       END_IF;
       RETURN;
   END_IF;

   IF (#tmpQuelle = 8) OR (#tmpQuelle = 12) THEN
       //Kurz rechts
       #Vorzug := NOT #Positionen[19].Sperre AND NOT #Positionen[20].Sperre AND #Positionen[23].Sperre AND NOT #Positionen[24].Sperre;

       IF NOT #Positionen[20].Sperre AND NOT #Vorzug THEN
           "FC_FW_Auftrag_Befehl"(inQuelle := #tmpQuelle,
                                  inZiel := 20,
                                  Befehl_ok => #Befehl_ok,
                                  outQuelle => #Quelle,
                                  outZiel => #Ziel);

           #nextStep := NOT #Befehl_ok;
       ELSIF NOT #Positionen[24].Sperre THEN
           "FC_FW_Auftrag_Befehl"(inQuelle := #tmpQuelle,
                                  inZiel := 24,
                                  Befehl_ok => #Befehl_ok,
                                  outQuelle => #Quelle,
                                  outZiel => #Ziel);

           #nextStep := NOT #Befehl_ok;
       ELSE
           #nextStep := TRUE;
       END_IF;
       RETURN;
   END_IF;

   //?
   #nextStep := TRUE;
END_REGION
END_FUNCTION

FUNCTION "FC_FW_Auftrag_Step4_KB" : Void   // FC1084, LAD
TITLE = Schritt WR02 -> CM03/CM04
{ S7_Optimized_Access := 'TRUE' }
// Ältesten Warenträger in WR02 suchen und nach CM03 / CM04 transportieren
// stored: AutoNumber false, SetENOAutomatically false
   VAR_INPUT
      Frg_Einfahrt : Bool;
      Frg_Schritt : Bool;
   END_VAR
   VAR_OUTPUT
      nextStep : Bool;
      startStep : Bool;
      parkStep : Bool;
   END_VAR
   VAR_IN_OUT
      Quelle : Int;
      Ziel : Int;
      Positionen : Array[1..30] of "UDT_Auftrag_Pos";
   END_VAR
   VAR_TEMP
      Sperre_Kurz_li_CM01 : Bool;
      Sperre_Kurz_li_CM02 : Bool;
      Sperre_Kurz_re_CM01 : Bool;
      Sperre_Kurz_re_CM02 : Bool;
      Sperre_Lang_CM01 : Bool;
      Sperre_Lang_CM02 : Bool;
      Vorzug : Bool;
      Befehl_ok : Bool;
      tmpQuelle : Int;
      Oldest : Real;
   END_VAR
BEGIN

REGION Network 1 (SCL)
   IF (#Quelle <> 0) AND (#Ziel <> 0) THEN
       #nextStep := #Positionen[#Quelle].Sperre;
       #startStep := NOT #nextStep;
       #Quelle := 0;
       #Ziel := 0;
       RETURN;
   END_IF;

   #Quelle := 0;
   #Ziel := 0;
   #nextStep := FALSE;
   #startStep := FALSE;

   IF NOT #Frg_Einfahrt OR NOT #Frg_Schritt THEN
       #nextStep := TRUE;
       RETURN;
   END_IF;
END_REGION

REGION Network 2 (SCL): Positionen sperren
   //Groß links nicht möglich - nur "161"
   #Positionen[27].CheckSperre := #Positionen[9].Sperre OR (#Positionen[3].Sperre);

   //Groß rechts nicht möglich
   #Positionen[28].CheckSperre := #Positionen[10].Sperre OR (#Positionen[4].Sperre);

   //kein Platz für Kurz links in CM03
   #Sperre_Kurz_li_CM01 := #Positionen[1].Sperre AND #Positionen[5].Sperre;
   #Sperre_Kurz_li_CM02 := #Positionen[13].Sperre AND #Positionen[17].Sperre;

   //kein Platz für Kurz rechts in CM03
   #Sperre_Kurz_re_CM01 := #Positionen[2].Sperre AND #Positionen[6].Sperre;
   #Sperre_Kurz_re_CM02 := #Positionen[14].Sperre AND #Positionen[18].Sperre;

   //kein Platz für Lang in CM03
   #Sperre_Lang_CM01 := ((#Positionen[1].Sperre OR #Positionen[2].Sperre) AND (#Positionen[5].Sperre OR #Positionen[6].Sperre));
   #Sperre_Lang_CM02 := ((#Positionen[13].Sperre OR #Positionen[14].Sperre) AND (#Positionen[17].Sperre OR #Positionen[18].Sperre));

   //Lang in P25 oder
   //kein Platz auf rechter Seite
   //-> P26 sperren
   #Positionen[26].CheckSperre := (#Positionen[26].WT_151 AND #Sperre_Kurz_re_CM02) OR (NOT #Positionen[26].WT_151 AND #Sperre_Kurz_re_CM01) OR (#Positionen[25].Wt_Typ = "WT_Typ_LS");

   //Lang in P25 und kein Platz für Lang oder
   //kein Platz auf linker Seite
   //-> P25 sperren
   IF #Positionen[25].WT_151 THEN
       #Positionen[25].CheckSperre := #Sperre_Kurz_li_CM02 OR ((#Positionen[25].Wt_Typ = "WT_Typ_LS") AND #Sperre_Lang_CM02);
   ELSE
       #Positionen[25].CheckSperre := #Sperre_Kurz_li_CM01 OR ((#Positionen[25].Wt_Typ = "WT_Typ_LS") AND #Sperre_Lang_CM01);
   END_IF;

   //Lang in P29 oder
   //kein Platz auf rechter Seite
   //-> P30 sperren
   #Positionen[30].CheckSperre := (#Positionen[30].WT_151 AND #Sperre_Kurz_re_CM02) OR (NOT #Positionen[30].WT_151 AND #Sperre_Kurz_re_CM01) OR (#Positionen[29].Wt_Typ = "WT_Typ_LS");

   //Lang in P29 und kein Platz für Lang oder
   //kein Platz auf linker Seite
   //-> P29 sperren
   IF #Positionen[29].WT_151 THEN
       #Positionen[29].CheckSperre := #Sperre_Kurz_li_CM02 OR ((#Positionen[29].Wt_Typ = "WT_Typ_LS") AND #Sperre_Lang_CM02);
   ELSE
       #Positionen[29].CheckSperre := #Sperre_Kurz_li_CM01 OR ((#Positionen[29].Wt_Typ = "WT_Typ_LS") AND #Sperre_Lang_CM01);
   END_IF;
END_REGION

REGION Network 3 (SCL): Ältesten WT suchen
   //
   #Oldest := 0;
   #tmpQuelle := 0;

   //WR02
   "FC_FW_Auftrag_Suche"(Pos1 := 25,
                         Pos2 := 30,
                         Positionen := #Positionen,
                         Quelle := #tmpQuelle,
                         Oldest := #Oldest);
END_REGION

REGION Network 4 (SCL): Auswertung
   IF #tmpQuelle = 0 THEN
       //kein WT
       #nextStep := TRUE;
       RETURN;
   END_IF;

   IF NOT #Positionen[#tmpQuelle].Fertig THEN
       #parkStep := TRUE;
       RETURN;
   END_IF;

   IF (#tmpQuelle = 27) THEN
       //Gross links - nur "161"
       IF NOT #Positionen[9].Sperre THEN
           "FC_FW_Auftrag_Befehl"(inQuelle := #tmpQuelle,
                                  inZiel := 9,
                                  Befehl_ok => #Befehl_ok,
                                  outQuelle => #Quelle,
                                  outZiel => #Ziel);

           #nextStep := NOT #Befehl_ok;
       ELSE
           #nextStep := TRUE;
       END_IF;
       RETURN;
   END_IF;

   IF (#tmpQuelle = 28) THEN
       //Gross rechts - nur "161"
       IF NOT #Positionen[10].Sperre THEN
           "FC_FW_Auftrag_Befehl"(inQuelle := #tmpQuelle,
                                  inZiel := 10,
                                  Befehl_ok => #Befehl_ok,
                                  outQuelle => #Quelle,
                                  outZiel => #Ziel);

           #nextStep := NOT #Befehl_ok;
       ELSE
           #nextStep := TRUE;
       END_IF;
       RETURN;
   END_IF;

   IF (#Positionen[#tmpQuelle].Wt_Typ = "WT_Typ_LS") AND ((#tmpQuelle = 25) OR (#tmpQuelle = 29)) AND NOT #Positionen[#tmpQuelle].WT_151 THEN
       //Lang "161"
       IF NOT #Positionen[11].Sperre AND NOT #Positionen[12].Sperre THEN
           "FC_FW_Auftrag_Befehl"(inQuelle := #tmpQuelle,
                                  inZiel := 11,
                                  Befehl_ok => #Befehl_ok,
                                  outQuelle => #Quelle,
                                  outZiel => #Ziel);

           #nextStep := NOT #Befehl_ok;
       ELSIF NOT #Positionen[7].Sperre AND NOT #Positionen[8].Sperre THEN
           "FC_FW_Auftrag_Befehl"(inQuelle := #tmpQuelle,
                                  inZiel := 7,
                                  Befehl_ok => #Befehl_ok,
                                  outQuelle => #Quelle,
                                  outZiel => #Ziel);

           #nextStep := NOT #Befehl_ok;
       ELSE
           #nextStep := TRUE;
       END_IF;
       RETURN;
   END_IF;

   IF (#Positionen[#tmpQuelle].Wt_Typ = "WT_Typ_LS") AND ((#tmpQuelle = 25) OR (#tmpQuelle = 29)) AND #Positionen[#tmpQuelle].WT_151 THEN
       //Lang "151"
       IF NOT #Positionen[23].Sperre AND NOT #Positionen[24].Sperre THEN
           "FC_FW_Auftrag_Befehl"(inQuelle := #tmpQuelle,
                                  inZiel := 23,
                                  Befehl_ok => #Befehl_ok,
                                  outQuelle => #Quelle,
                                  outZiel => #Ziel);

           #nextStep := NOT #Befehl_ok;
       ELSIF NOT #Positionen[19].Sperre AND NOT #Positionen[20].Sperre THEN
           "FC_FW_Auftrag_Befehl"(inQuelle := #tmpQuelle,
                                  inZiel := 19,
                                  Befehl_ok => #Befehl_ok,
                                  outQuelle => #Quelle,
                                  outZiel => #Ziel);

           #nextStep := NOT #Befehl_ok;
       ELSE
           #nextStep := TRUE;
       END_IF;
       RETURN;
   END_IF;


   IF ((#tmpQuelle = 25) OR (#tmpQuelle = 29)) AND NOT #Positionen[#tmpQuelle].WT_151 THEN
       //Kurz links "161"
       #Vorzug := NOT #Positionen[11].Sperre AND NOT #Positionen[12].Sperre AND NOT #Positionen[7].Sperre AND #Positionen[8].Sperre;

       IF NOT #Positionen[11].Sperre AND NOT #Vorzug THEN
           "FC_FW_Auftrag_Befehl"(inQuelle := #tmpQuelle,
                                  inZiel := 11,
                                  Befehl_ok => #Befehl_ok,
                                  outQuelle => #Quelle,
                                  outZiel => #Ziel);

           #nextStep := NOT #Befehl_ok;
       ELSIF NOT #Positionen[7].Sperre THEN
           "FC_FW_Auftrag_Befehl"(inQuelle := #tmpQuelle,
                                  inZiel := 7,
                                  Befehl_ok => #Befehl_ok,
                                  outQuelle => #Quelle,
                                  outZiel => #Ziel);

           #nextStep := NOT #Befehl_ok;
       ELSE
           #nextStep := TRUE;
       END_IF;
       RETURN;
   END_IF;

   IF ((#tmpQuelle = 26) OR (#tmpQuelle = 30)) AND NOT #Positionen[#tmpQuelle].WT_151 THEN
       //Kurz rechts "161"
       #Vorzug := NOT #Positionen[11].Sperre AND NOT #Positionen[12].Sperre AND #Positionen[7].Sperre AND NOT #Positionen[8].Sperre;

       IF NOT #Positionen[12].Sperre AND NOT #Vorzug THEN
           "FC_FW_Auftrag_Befehl"(inQuelle := #tmpQuelle,
                                  inZiel := 12,
                                  Befehl_ok => #Befehl_ok,
                                  outQuelle => #Quelle,
                                  outZiel => #Ziel);

           #nextStep := NOT #Befehl_ok;
       ELSIF NOT #Positionen[8].Sperre THEN
           "FC_FW_Auftrag_Befehl"(inQuelle := #tmpQuelle,
                                  inZiel := 8,
                                  Befehl_ok => #Befehl_ok,
                                  outQuelle => #Quelle,
                                  outZiel => #Ziel);

           #nextStep := NOT #Befehl_ok;
       ELSE
           #nextStep := TRUE;
       END_IF;
       RETURN;
   END_IF;


   IF ((#tmpQuelle = 25) OR (#tmpQuelle = 29)) AND #Positionen[#tmpQuelle].WT_151 THEN
       //Kurz links "151"
       #Vorzug := NOT #Positionen[23].Sperre AND NOT #Positionen[24].Sperre AND NOT #Positionen[19].Sperre AND #Positionen[20].Sperre;

       IF NOT #Positionen[23].Sperre AND NOT #Vorzug THEN
           "FC_FW_Auftrag_Befehl"(inQuelle := #tmpQuelle,
                                  inZiel := 23,
                                  Befehl_ok => #Befehl_ok,
                                  outQuelle => #Quelle,
                                  outZiel => #Ziel);

           #nextStep := NOT #Befehl_ok;
       ELSIF NOT #Positionen[19].Sperre THEN
           "FC_FW_Auftrag_Befehl"(inQuelle := #tmpQuelle,
                                  inZiel := 19,
                                  Befehl_ok => #Befehl_ok,
                                  outQuelle => #Quelle,
                                  outZiel => #Ziel);

           #nextStep := NOT #Befehl_ok;
       ELSE
           #nextStep := TRUE;
       END_IF;
       RETURN;
   END_IF;

   IF ((#tmpQuelle = 26) OR (#tmpQuelle = 30)) AND  #Positionen[#tmpQuelle].WT_151 THEN
       //Kurz rechts "151"
       #Vorzug := NOT #Positionen[23].Sperre AND NOT #Positionen[24].Sperre AND #Positionen[23].Sperre AND NOT #Positionen[24].Sperre;

       IF NOT #Positionen[24].Sperre AND NOT #Vorzug THEN
           "FC_FW_Auftrag_Befehl"(inQuelle := #tmpQuelle,
                                  inZiel := 24,
                                  Befehl_ok => #Befehl_ok,
                                  outQuelle => #Quelle,
                                  outZiel => #Ziel);

           #nextStep := NOT #Befehl_ok;
       ELSIF NOT #Positionen[20].Sperre THEN
           "FC_FW_Auftrag_Befehl"(inQuelle := #tmpQuelle,
                                  inZiel := 20,
                                  Befehl_ok => #Befehl_ok,
                                  outQuelle => #Quelle,
                                  outZiel => #Ziel);

           #nextStep := NOT #Befehl_ok;
       ELSE
           #nextStep := TRUE;
       END_IF;
       RETURN;
   END_IF;

   //
   #nextStep := TRUE;
END_REGION
END_FUNCTION

FUNCTION "FC_FW_Auftrag_Step4_NB" : Void   // FC184, LAD
TITLE = Schritt WR02 -> CM03
{ S7_Optimized_Access := 'TRUE' }
// Ältesten Warenträger in WR02 suchen und nach CM03 transportieren
// stored: AutoNumber false, SetENOAutomatically false
   VAR_INPUT
      Frg_Einfahrt : Bool;
      Frg_Schritt : Bool;
   END_VAR
   VAR_OUTPUT
      nextStep : Bool;
      startStep : Bool;
      parkStep : Bool;
   END_VAR
   VAR_IN_OUT
      Quelle : Int;
      Ziel : Int;
      Positionen : Array[1..30] of "UDT_Auftrag_Pos";
   END_VAR
   VAR_TEMP
      Sperre_Kurz_li : Bool;
      Sperre_Kurz_li_CM01 : Bool;
      Sperre_Kurz_li_CM02 : Bool;
      Sperre_Kurz_re : Bool;
      Sperre_Kurz_re_CM01 : Bool;
      Sperre_Kurz_re_CM02 : Bool;
      Sperre_Lang : Bool;
      Sperre_Lang_CM01 : Bool;
      Sperre_Lang_CM02 : Bool;
      Vorzug : Bool;
      Befehl_ok : Bool;
      tmpQuelle : Int;
      Oldest : Real;
   END_VAR
BEGIN

REGION Network 1 (SCL)
   IF (#Quelle <> 0) AND (#Ziel <> 0) THEN
       #nextStep := #Positionen[#Quelle].Sperre;
       #startStep := NOT #nextStep;
       #Quelle := 0;
       #Ziel := 0;
       RETURN;
   END_IF;

   #Quelle := 0;
   #Ziel := 0;
   #nextStep := FALSE;
   #startStep := FALSE;

   IF NOT #Frg_Einfahrt OR NOT #Frg_Schritt THEN
       #nextStep := TRUE;
       RETURN;
   END_IF;
END_REGION

REGION Network 2 (SCL): Positionen sperren
   //Groß links nicht möglich
   #Positionen[27].CheckSperre := #Positionen[9].Sperre OR (#Positionen[3].Sperre AND #Positionen[15].Sperre);

   //Groß rechts nicht möglich
   #Positionen[28].CheckSperre := #Positionen[10].Sperre OR (#Positionen[4].Sperre AND #Positionen[16].Sperre);

   //kein Platz für Kurz links in CM03
   #Sperre_Kurz_li_CM01 := #Positionen[1].Sperre AND #Positionen[5].Sperre;
   #Sperre_Kurz_li_CM02 := #Positionen[13].Sperre AND #Positionen[17].Sperre;
   #Sperre_Kurz_li := (#Positionen[7].Sperre AND #Positionen[11].Sperre) OR (#Sperre_Kurz_li_CM01 AND #Sperre_Kurz_li_CM02);

   //kein Platz für Kurz rechts in CM03
   #Sperre_Kurz_re_CM01 := #Positionen[2].Sperre AND #Positionen[6].Sperre;
   #Sperre_Kurz_re_CM02 := #Positionen[14].Sperre AND #Positionen[18].Sperre;
   #Sperre_Kurz_re := (#Positionen[8].Sperre AND #Positionen[12].Sperre) OR (#Sperre_Kurz_re_CM01 AND #Sperre_Kurz_re_CM02);

   //kein Platz für Lang in CM03
   #Sperre_Lang_CM01 := ((#Positionen[1].Sperre OR #Positionen[2].Sperre) AND (#Positionen[5].Sperre OR #Positionen[6].Sperre));
   #Sperre_Lang_CM02 := ((#Positionen[13].Sperre OR #Positionen[14].Sperre) AND (#Positionen[17].Sperre OR #Positionen[18].Sperre));
   #Sperre_Lang := ((#Positionen[7].Sperre OR #Positionen[8].Sperre) AND (#Positionen[11].Sperre OR #Positionen[12].Sperre)) OR (#Sperre_Lang_CM01 AND #Sperre_Lang_CM02);

   //Lang in P25 oder
   //kein Platz auf rechter Seite
   //-> P26 sperren
   #Positionen[26].CheckSperre := #Sperre_Kurz_re OR (#Positionen[25].Wt_Typ = "WT_Typ_LS");

   //Lang in P25 und kein Platz für Lang oder
   //kein Platz auf linker Seite
   //-> P25 sperren
   #Positionen[25].CheckSperre := #Sperre_Kurz_li OR ((#Positionen[25].Wt_Typ = "WT_Typ_LS") AND #Sperre_Lang);

   //Lang in P29 oder
   //kein Platz auf rechter Seite
   //-> P30 sperren
   #Positionen[30].CheckSperre := #Sperre_Kurz_re OR (#Positionen[29].Wt_Typ = "WT_Typ_LS");

   //Lang in P29 und kein Platz für Lang oder
   //kein Platz auf linker Seite
   //-> P29 sperren
   #Positionen[29].CheckSperre := #Sperre_Kurz_li OR ((#Positionen[29].Wt_Typ = "WT_Typ_LS") AND #Sperre_Lang);
END_REGION

REGION Network 3 (SCL): Ältesten WT suchen
   //
   #Oldest := 0;
   #tmpQuelle := 0;

   //WR02
   "FC_FW_Auftrag_Suche"(Pos1 := 25,
                         Pos2 := 30,
                         Positionen := #Positionen,
                         Quelle := #tmpQuelle,
                         Oldest := #Oldest);
END_REGION

REGION Network 4 (SCL): Auswertung
   IF #tmpQuelle = 0 THEN
       //kein WT
       #nextStep := TRUE;
       RETURN;
   END_IF;

   IF NOT #Positionen[#tmpQuelle].Fertig THEN
       #parkStep := TRUE;
       RETURN;
   END_IF;

   IF (#tmpQuelle = 27) THEN
       //Gross links
       IF NOT #Positionen[9].Sperre THEN
           "FC_FW_Auftrag_Befehl"(inQuelle := #tmpQuelle,
                                  inZiel := 9,
                                  Befehl_ok => #Befehl_ok,
                                  outQuelle => #Quelle,
                                  outZiel => #Ziel);

           #nextStep := NOT #Befehl_ok;
       ELSE
           #nextStep := TRUE;
       END_IF;
       RETURN;
   END_IF;

   IF (#tmpQuelle = 28) THEN
       //Gross rechts
       IF NOT #Positionen[10].Sperre THEN
           "FC_FW_Auftrag_Befehl"(inQuelle := #tmpQuelle,
                                  inZiel := 10,
                                  Befehl_ok => #Befehl_ok,
                                  outQuelle => #Quelle,
                                  outZiel => #Ziel);

           #nextStep := NOT #Befehl_ok;
       ELSE
           #nextStep := TRUE;
       END_IF;
       RETURN;
   END_IF;

   IF (#Positionen[#tmpQuelle].Wt_Typ = "WT_Typ_LS") AND ((#tmpQuelle = 25) OR (#tmpQuelle = 29)) THEN
       //Lang
       IF NOT #Positionen[11].Sperre AND NOT #Positionen[12].Sperre THEN
           "FC_FW_Auftrag_Befehl"(inQuelle := #tmpQuelle,
                                  inZiel := 11,
                                  Befehl_ok => #Befehl_ok,
                                  outQuelle => #Quelle,
                                  outZiel => #Ziel);

           #nextStep := NOT #Befehl_ok;
       ELSIF NOT #Positionen[7].Sperre AND NOT #Positionen[8].Sperre THEN
           "FC_FW_Auftrag_Befehl"(inQuelle := #tmpQuelle,
                                  inZiel := 7,
                                  Befehl_ok => #Befehl_ok,
                                  outQuelle => #Quelle,
                                  outZiel => #Ziel);

           #nextStep := NOT #Befehl_ok;
       ELSE
           #nextStep := TRUE;
       END_IF;
       RETURN;
   END_IF;

   IF (#tmpQuelle = 25) OR (#tmpQuelle = 29) THEN
       //Kurz links
       #Vorzug := NOT #Positionen[11].Sperre AND NOT #Positionen[12].Sperre AND NOT #Positionen[7].Sperre AND #Positionen[8].Sperre;

       IF NOT #Positionen[11].Sperre AND NOT #Vorzug THEN
           "FC_FW_Auftrag_Befehl"(inQuelle := #tmpQuelle,
                                  inZiel := 11,
                                  Befehl_ok => #Befehl_ok,
                                  outQuelle => #Quelle,
                                  outZiel => #Ziel);

           #nextStep := NOT #Befehl_ok;
       ELSIF NOT #Positionen[7].Sperre THEN
           "FC_FW_Auftrag_Befehl"(inQuelle := #tmpQuelle,
                                  inZiel := 7,
                                  Befehl_ok => #Befehl_ok,
                                  outQuelle => #Quelle,
                                  outZiel => #Ziel);

           #nextStep := NOT #Befehl_ok;
       ELSE
           #nextStep := TRUE;
       END_IF;
       RETURN;
   END_IF;

   IF (#tmpQuelle = 26) OR (#tmpQuelle = 30) THEN
       //Kurz rechts
       #Vorzug := NOT #Positionen[11].Sperre AND NOT #Positionen[12].Sperre AND #Positionen[7].Sperre AND NOT #Positionen[8].Sperre;

       IF NOT #Positionen[12].Sperre AND NOT #Vorzug THEN
           "FC_FW_Auftrag_Befehl"(inQuelle := #tmpQuelle,
                                  inZiel := 12,
                                  Befehl_ok => #Befehl_ok,
                                  outQuelle => #Quelle,
                                  outZiel => #Ziel);

           #nextStep := NOT #Befehl_ok;
       ELSIF NOT #Positionen[8].Sperre THEN
           "FC_FW_Auftrag_Befehl"(inQuelle := #tmpQuelle,
                                  inZiel := 8,
                                  Befehl_ok => #Befehl_ok,
                                  outQuelle => #Quelle,
                                  outZiel => #Ziel);

           #nextStep := NOT #Befehl_ok;
       ELSE
           #nextStep := TRUE;
       END_IF;
       RETURN;
   END_IF;

   //?
   #nextStep := TRUE;
END_REGION
END_FUNCTION

FUNCTION "FC_FW_Auftrag_Step5_KB" : Void   // FC1085, LAD
TITLE = Schritt CM03/CM04 -> WR02
{ S7_Optimized_Access := 'TRUE' }
// Ältesten Warenträger in CM03/CM04 suchen und nach WR02 transportieren
// stored: AutoNumber false, SetENOAutomatically false
   VAR_INPUT
      Frg_Schritt : Bool;
   END_VAR
   VAR_OUTPUT
      nextStep : Bool;
      startStep : Bool;
      parkStep : Bool;
   END_VAR
   VAR_IN_OUT
      Quelle : Int;
      Ziel : Int;
      Positionen : Array[1..30] of "UDT_Auftrag_Pos";
      Frg_Ausfahrt : Bool;
   END_VAR
   VAR_TEMP
      Sperre_Kurz_li : Bool;
      Sperre_Kurz_re : Bool;
      Sperre_Lang : Bool;
      Vorzug : Bool;
      Befehl_ok : Bool;
      tmpQuelle : Int;
      Oldest : Real;
   END_VAR
   VAR CONSTANT
      Wt_Cmd_Ausfahrt : Int := 25;
   END_VAR
BEGIN

REGION Network 1 (SCL)
   IF (#Quelle <> 0) AND (#Ziel <> 0) THEN
       #nextStep := #Positionen[#Quelle].Sperre;
       #startStep := NOT #nextStep;
       #Quelle := 0;
       #Ziel := 0;
       #Frg_Ausfahrt := NOT #startStep;
       RETURN;
   END_IF;

   #Quelle := 0;
   #Ziel := 0;
   #nextStep := FALSE;
   #startStep := FALSE;
END_REGION

REGION Network 2 (SCL): Anmeldung Großoptik
   //alle Positionen suchbar
   #Positionen[7].CheckSperre := FALSE;
   #Positionen[8].CheckSperre := FALSE;
   #Positionen[9].CheckSperre := FALSE;
   #Positionen[10].CheckSperre := FALSE;
   #Positionen[11].CheckSperre := FALSE;
   #Positionen[12].CheckSperre := FALSE;

   #Positionen[19].CheckSperre := FALSE;
   #Positionen[20].CheckSperre := FALSE;
   #Positionen[21].CheckSperre := FALSE;
   #Positionen[22].CheckSperre := FALSE;
   #Positionen[23].CheckSperre := FALSE;
   #Positionen[24].CheckSperre := FALSE;

   //
   #Oldest := 0;
   #tmpQuelle := 0;

   //CM03
   "FC_FW_Auftrag_Suche"(Pos1 := 7,
                         Pos2 := 12,
                         Positionen := #Positionen,
                         Quelle := #tmpQuelle,
                         Oldest := #Oldest);

   //CM04
   "FC_FW_Auftrag_Suche"(Pos1 := 19,
                         Pos2 := 24,
                         Positionen := #Positionen,
                         Quelle := #tmpQuelle,
                         Oldest := #Oldest);

   IF ((#tmpQuelle = 9) OR (#tmpQuelle = 10)) AND #Frg_Ausfahrt AND #Frg_Schritt THEN
       //Großoptik ist ältester
       #Vorzug := NOT "DI_QF_WR02_03".In.Req_Ausfahrt_GO;
       "DI_QF_WR02_03".In.Req_Ausfahrt_GO := TRUE;
   ELSE
       #Vorzug := FALSE;
       "DI_QF_WR02_03".In.Req_Ausfahrt_GO := FALSE;
   END_IF;

   IF (#tmpQuelle = 0) OR NOT #Frg_Schritt THEN
       #Frg_Ausfahrt := FALSE;
   END_IF;
END_REGION

REGION Network 3 (SCL): Positionen sperren
   IF NOT #Frg_Ausfahrt OR NOT #Frg_Schritt THEN
       #nextStep := TRUE;
       RETURN;
   END_IF;

   // GO nur "161" (CM03)

   //Groß links nicht möglich
   #Positionen[9].CheckSperre := #Positionen[27].Sperre OR (#Positionen[9].Wt_Cmd <> #Wt_Cmd_Ausfahrt);

   //Groß rechts nicht möglich
   #Positionen[10].CheckSperre := #Positionen[28].Sperre OR (#Positionen[10].Wt_Cmd <> #Wt_Cmd_Ausfahrt);

   //kein Platz für Kurz links in WR02
   #Sperre_Kurz_li := (#Positionen[25].Sperre AND #Positionen[29].Sperre) OR #Vorzug;

   //kein Platz für Kurz rechts in WR02
   #Sperre_Kurz_re := (#Positionen[26].Sperre AND #Positionen[30].Sperre) OR #Vorzug;

   //kein Platz für Lang in WR02
   #Sperre_Lang := ((#Positionen[25].Sperre OR #Positionen[26].Sperre) AND (#Positionen[29].Sperre OR #Positionen[30].Sperre)) OR #Vorzug;

   // "151" CM04
   //Lang in P19 oder
   //kein Platz auf rechter Seite
   //-> P20 sperren
   #Positionen[20].CheckSperre := #Sperre_Kurz_re OR (#Positionen[19].Wt_Typ = "WT_Typ_LS") OR (#Positionen[20].Wt_Cmd <> #Wt_Cmd_Ausfahrt);

   //Lang in P19 und kein Platz für Lang oder
   //kein Platz auf linker Seite
   //-> P19 sperren
   #Positionen[19].CheckSperre := #Sperre_Kurz_li OR ((#Positionen[19].Wt_Typ = "WT_Typ_LS") AND #Sperre_Lang) OR (#Positionen[19].Wt_Cmd <> #Wt_Cmd_Ausfahrt);

   //Lang in P23 oder
   //kein Platz auf rechter Seite
   //-> P24 sperren
   #Positionen[24].CheckSperre := #Sperre_Kurz_re OR (#Positionen[23].Wt_Typ = "WT_Typ_LS") OR (#Positionen[24].Wt_Cmd <> #Wt_Cmd_Ausfahrt);

   //Lang in P23 und kein Platz für Lang oder
   //kein Platz auf linker Seite
   //-> P23 sperren
   #Positionen[23].CheckSperre := #Sperre_Kurz_li OR ((#Positionen[23].Wt_Typ = "WT_Typ_LS") AND #Sperre_Lang) OR (#Positionen[23].Wt_Cmd <> #Wt_Cmd_Ausfahrt);

   // "161" CM03
   //Lang in P7 oder
   //kein Platz auf rechter Seite
   //-> P8 sperren
   #Positionen[8].CheckSperre := #Sperre_Kurz_re OR (#Positionen[7].Wt_Typ = "WT_Typ_LS") OR (#Positionen[8].Wt_Cmd <> #Wt_Cmd_Ausfahrt);

   //Lang in P7 und kein Platz für Lang oder
   //kein Platz auf linker Seite
   //-> P7 sperren
   #Positionen[7].CheckSperre := #Sperre_Kurz_li OR ((#Positionen[7].Wt_Typ = "WT_Typ_LS") AND #Sperre_Lang) OR (#Positionen[7].Wt_Cmd <> #Wt_Cmd_Ausfahrt);

   //Lang in P11 oder
   //kein Platz auf rechter Seite
   //-> P12 sperren
   #Positionen[12].CheckSperre := #Sperre_Kurz_re OR (#Positionen[11].Wt_Typ = "WT_Typ_LS") OR (#Positionen[12].Wt_Cmd <> #Wt_Cmd_Ausfahrt);

   //Lang in P11 und kein Platz für Lang oder
   //kein Platz auf linker Seite
   //-> P23 sperren
   #Positionen[11].CheckSperre := #Sperre_Kurz_li OR ((#Positionen[11].Wt_Typ = "WT_Typ_LS") AND #Sperre_Lang) OR (#Positionen[11].Wt_Cmd <> #Wt_Cmd_Ausfahrt);
END_REGION

REGION Network 4 (SCL): Ältesten WT suchen
   //
   #Oldest := 0;
   #tmpQuelle := 0;

   //CM04
   "FC_FW_Auftrag_Suche"(Pos1 := 19,
                         Pos2 := 24,
                         Positionen := #Positionen,
                         Quelle := #tmpQuelle,
                         Oldest := #Oldest);

   //CM03
   "FC_FW_Auftrag_Suche"(Pos1 := 7,
                         Pos2 := 12,
                         Positionen := #Positionen,
                         Quelle := #tmpQuelle,
                         Oldest := #Oldest);
END_REGION

REGION Network 5 (SCL): Auswertung
   IF #tmpQuelle = 0 THEN
       //kein WT
       #nextStep := TRUE;
       RETURN;
   END_IF;

   IF NOT #Positionen[#tmpQuelle].Fertig THEN
       #parkStep := TRUE;
       RETURN;
   END_IF;

   // GO nur 161
   IF (#tmpQuelle = 9) THEN
       //Gross links
       IF NOT #Positionen[27].Sperre THEN
           "FC_FW_Auftrag_Befehl"(inQuelle := #tmpQuelle,
                                  inZiel := 27,
                                  Befehl_ok => #Befehl_ok,
                                  outQuelle => #Quelle,
                                  outZiel => #Ziel);

           #nextStep := NOT #Befehl_ok;
       ELSE
           #nextStep := TRUE;
       END_IF;
       RETURN;
   END_IF;

   IF (#tmpQuelle = 10) THEN
       //Gross rechts
       IF NOT #Positionen[28].Sperre THEN
           "FC_FW_Auftrag_Befehl"(inQuelle := #tmpQuelle,
                                  inZiel := 28,
                                  Befehl_ok => #Befehl_ok,
                                  outQuelle => #Quelle,
                                  outZiel => #Ziel);

           #nextStep := NOT #Befehl_ok;
       ELSE
           #nextStep := TRUE;
       END_IF;
       RETURN;
   END_IF;

   IF (#Positionen[#tmpQuelle].Wt_Typ = "WT_Typ_LS") AND ((#tmpQuelle = 19) OR (#tmpQuelle = 23) OR (#tmpQuelle = 7)OR (#tmpQuelle = 11) )THEN
       //Lang
       IF NOT #Positionen[25].Sperre AND NOT #Positionen[26].Sperre THEN
           "FC_FW_Auftrag_Befehl"(inQuelle := #tmpQuelle,
                                  inZiel := 25,
                                  Befehl_ok => #Befehl_ok,
                                  outQuelle => #Quelle,
                                  outZiel => #Ziel);

           #nextStep := NOT #Befehl_ok;
       ELSIF NOT #Positionen[29].Sperre AND NOT #Positionen[30].Sperre THEN
           "FC_FW_Auftrag_Befehl"(inQuelle := #tmpQuelle,
                                  inZiel := 29,
                                  Befehl_ok => #Befehl_ok,
                                  outQuelle => #Quelle,
                                  outZiel => #Ziel);

           #nextStep := NOT #Befehl_ok;
       ELSE
           #nextStep := TRUE;
       END_IF;
       RETURN;
   END_IF;

   IF (#tmpQuelle = 19) OR (#tmpQuelle = 23) OR (#tmpQuelle = 7) OR (#tmpQuelle = 11) THEN
       //Kurz links
       #Vorzug := NOT #Positionen[25].Sperre AND NOT #Positionen[26].Sperre AND NOT #Positionen[29].Sperre AND #Positionen[30].Sperre;

       IF NOT #Positionen[25].Sperre AND NOT #Vorzug THEN
           "FC_FW_Auftrag_Befehl"(inQuelle := #tmpQuelle,
                                  inZiel := 25,
                                  Befehl_ok => #Befehl_ok,
                                  outQuelle => #Quelle,
                                  outZiel => #Ziel);

           #nextStep := NOT #Befehl_ok;
       ELSIF NOT #Positionen[29].Sperre THEN
           "FC_FW_Auftrag_Befehl"(inQuelle := #tmpQuelle,
                                  inZiel := 29,
                                  Befehl_ok => #Befehl_ok,
                                  outQuelle => #Quelle,
                                  outZiel => #Ziel);

           #nextStep := NOT #Befehl_ok;
       ELSE
           #nextStep := TRUE;
       END_IF;
       RETURN;
   END_IF;

   IF (#tmpQuelle = 20) OR (#tmpQuelle = 24) OR (#tmpQuelle = 8) OR (#tmpQuelle = 12) THEN
       //Kurz rechts
       #Vorzug := NOT #Positionen[25].Sperre AND NOT #Positionen[26].Sperre AND #Positionen[29].Sperre AND NOT #Positionen[30].Sperre;

       IF NOT #Positionen[26].Sperre AND NOT #Vorzug THEN
           "FC_FW_Auftrag_Befehl"(inQuelle := #tmpQuelle,
                                  inZiel := 26,
                                  Befehl_ok => #Befehl_ok,
                                  outQuelle => #Quelle,
                                  outZiel => #Ziel);

           #nextStep := NOT #Befehl_ok;
       ELSIF NOT #Positionen[30].Sperre THEN
           "FC_FW_Auftrag_Befehl"(inQuelle := #tmpQuelle,
                                  inZiel := 30,
                                  Befehl_ok => #Befehl_ok,
                                  outQuelle => #Quelle,
                                  outZiel => #Ziel);

           #nextStep := NOT #Befehl_ok;
       ELSE
           #nextStep := TRUE;
       END_IF;
       RETURN;
   END_IF;

   //
   #nextStep := TRUE;
END_REGION
END_FUNCTION

FUNCTION "FC_FW_Auftrag_Step5_NB" : Void   // FC185, LAD
TITLE = Schritt CM04 -> WR02
{ S7_Optimized_Access := 'TRUE' }
// Ältesten Warenträger in CM04 suchen und nach WR02 transportieren
// stored: AutoNumber false, SetENOAutomatically false
   VAR_INPUT
      Frg_Schritt : Bool;
   END_VAR
   VAR_OUTPUT
      nextStep : Bool;
      startStep : Bool;
      parkStep : Bool;
   END_VAR
   VAR_IN_OUT
      Quelle : Int;
      Ziel : Int;
      Positionen : Array[1..30] of "UDT_Auftrag_Pos";
      Frg_Ausfahrt : Bool;
   END_VAR
   VAR_TEMP
      Sperre_Kurz_li : Bool;
      Sperre_Kurz_re : Bool;
      Sperre_Lang : Bool;
      Vorzug : Bool;
      Befehl_ok : Bool;
      tmpQuelle : Int;
      Oldest : Real;
   END_VAR
BEGIN

REGION Network 1 (SCL)
   IF (#Quelle <> 0) AND (#Ziel <> 0) THEN
       #nextStep := #Positionen[#Quelle].Sperre;
       #startStep := NOT #nextStep;
       #Quelle := 0;
       #Ziel := 0;
       #Frg_Ausfahrt := NOT #startStep;
       RETURN;
   END_IF;

   #Quelle := 0;
   #Ziel := 0;
   #nextStep := FALSE;
   #startStep := FALSE;
END_REGION

REGION Network 2 (SCL): Anmeldung Großoptik
   //alle Positionen suchbar
   #Positionen[19].CheckSperre := FALSE;
   #Positionen[20].CheckSperre := FALSE;
   #Positionen[21].CheckSperre := FALSE;
   #Positionen[22].CheckSperre := FALSE;
   #Positionen[23].CheckSperre := FALSE;
   #Positionen[24].CheckSperre := FALSE;

   //
   #Oldest := 0;
   #tmpQuelle := 0;

   //CM04
   "FC_FW_Auftrag_Suche"(Pos1 := 19,
                         Pos2 := 24,
                         Positionen := #Positionen,
                         Quelle := #tmpQuelle,
                         Oldest := #Oldest);

   IF ((#tmpQuelle = 21) OR (#tmpQuelle = 22)) AND #Frg_Ausfahrt AND #Frg_Schritt THEN
       //Großoptik ist ältester
       #Vorzug := NOT "DI_QF_WR02_03".In.Req_Ausfahrt_GO;
       "DI_QF_WR02_03".In.Req_Ausfahrt_GO := TRUE;
   ELSE
       #Vorzug := FALSE;
       "DI_QF_WR02_03".In.Req_Ausfahrt_GO := FALSE;
   END_IF;

   IF (#tmpQuelle = 0) OR NOT #Frg_Schritt THEN
       #Frg_Ausfahrt := FALSE;
   END_IF;
END_REGION

REGION Network 3 (SCL): Positionen sperren
   IF NOT #Frg_Ausfahrt OR NOT #Frg_Schritt THEN
       #nextStep := TRUE;
       RETURN;
   END_IF;

   //Groß links nicht möglich
   #Positionen[21].CheckSperre := #Positionen[27].Sperre;

   //Groß rechts nicht möglich
   #Positionen[22].CheckSperre := #Positionen[28].Sperre;

   //kein Platz für Kurz links in WR02
   #Sperre_Kurz_li := (#Positionen[25].Sperre AND #Positionen[29].Sperre) OR #Vorzug;

   //kein Platz für Kurz rechts in WR02
   #Sperre_Kurz_re := (#Positionen[26].Sperre AND #Positionen[30].Sperre) OR #Vorzug;

   //kein Platz für Lang in WR02
   #Sperre_Lang := ((#Positionen[25].Sperre OR #Positionen[26].Sperre) AND (#Positionen[29].Sperre OR #Positionen[30].Sperre)) OR #Vorzug;

   //Lang in P19 oder
   //kein Platz auf rechter Seite
   //-> P20 sperren
   #Positionen[20].CheckSperre := #Sperre_Kurz_re OR (#Positionen[19].Wt_Typ = "WT_Typ_LS");

   //Lang in P19 und kein Platz für Lang oder
   //kein Platz auf linker Seite
   //-> P19 sperren
   #Positionen[19].CheckSperre := #Sperre_Kurz_li OR ((#Positionen[19].Wt_Typ = "WT_Typ_LS") AND #Sperre_Lang);

   //Lang in P23 oder
   //kein Platz auf rechter Seite
   //-> P24 sperren
   #Positionen[24].CheckSperre := #Sperre_Kurz_re OR (#Positionen[23].Wt_Typ = "WT_Typ_LS");

   //Lang in P23 und kein Platz für Lang oder
   //kein Platz auf linker Seite
   //-> P23 sperren
   #Positionen[23].CheckSperre := #Sperre_Kurz_li OR ((#Positionen[23].Wt_Typ = "WT_Typ_LS") AND #Sperre_Lang);
END_REGION

REGION Network 4 (SCL): Ältesten WT suchen
   //
   #Oldest := 0;
   #tmpQuelle := 0;

   //CM04
   "FC_FW_Auftrag_Suche"(Pos1 := 19,
                         Pos2 := 24,
                         Positionen := #Positionen,
                         Quelle := #tmpQuelle,
                         Oldest := #Oldest);
END_REGION

REGION Network 5 (SCL): Auswertung
   IF #tmpQuelle = 0 THEN
       //kein WT
       #nextStep := TRUE;
       RETURN;
   END_IF;

   IF NOT #Positionen[#tmpQuelle].Fertig THEN
       #parkStep := TRUE;
       RETURN;
   END_IF;

   IF (#tmpQuelle = 21) THEN
       //Gross links
       IF NOT #Positionen[27].Sperre THEN
           "FC_FW_Auftrag_Befehl"(inQuelle := #tmpQuelle,
                                  inZiel := 27,
                                  Befehl_ok => #Befehl_ok,
                                  outQuelle => #Quelle,
                                  outZiel => #Ziel);

           #nextStep := NOT #Befehl_ok;
       ELSE
           #nextStep := TRUE;
       END_IF;
       RETURN;
   END_IF;

   IF (#tmpQuelle = 22) THEN
       //Gross rechts
       IF NOT #Positionen[28].Sperre THEN
           "FC_FW_Auftrag_Befehl"(inQuelle := #tmpQuelle,
                                  inZiel := 28,
                                  Befehl_ok => #Befehl_ok,
                                  outQuelle => #Quelle,
                                  outZiel => #Ziel);

           #nextStep := NOT #Befehl_ok;
       ELSE
           #nextStep := TRUE;
       END_IF;
       RETURN;
   END_IF;

   IF (#Positionen[#tmpQuelle].Wt_Typ = "WT_Typ_LS") AND ((#tmpQuelle = 19) OR (#tmpQuelle = 23)) THEN
       //Lang
       IF NOT #Positionen[25].Sperre AND NOT #Positionen[26].Sperre THEN
           "FC_FW_Auftrag_Befehl"(inQuelle := #tmpQuelle,
                                  inZiel := 25,
                                  Befehl_ok => #Befehl_ok,
                                  outQuelle => #Quelle,
                                  outZiel => #Ziel);

           #nextStep := NOT #Befehl_ok;
       ELSIF NOT #Positionen[29].Sperre AND NOT #Positionen[30].Sperre THEN
           "FC_FW_Auftrag_Befehl"(inQuelle := #tmpQuelle,
                                  inZiel := 29,
                                  Befehl_ok => #Befehl_ok,
                                  outQuelle => #Quelle,
                                  outZiel => #Ziel);

           #nextStep := NOT #Befehl_ok;
       ELSE
           #nextStep := TRUE;
       END_IF;
       RETURN;
   END_IF;

   IF (#tmpQuelle = 19) OR (#tmpQuelle = 23) THEN
       //Kurz links
       #Vorzug := NOT #Positionen[25].Sperre AND NOT #Positionen[26].Sperre AND NOT #Positionen[29].Sperre AND #Positionen[30].Sperre;

       IF NOT #Positionen[25].Sperre AND NOT #Vorzug THEN
           "FC_FW_Auftrag_Befehl"(inQuelle := #tmpQuelle,
                                  inZiel := 25,
                                  Befehl_ok => #Befehl_ok,
                                  outQuelle => #Quelle,
                                  outZiel => #Ziel);

           #nextStep := NOT #Befehl_ok;
       ELSIF NOT #Positionen[29].Sperre THEN
           "FC_FW_Auftrag_Befehl"(inQuelle := #tmpQuelle,
                                  inZiel := 29,
                                  Befehl_ok => #Befehl_ok,
                                  outQuelle => #Quelle,
                                  outZiel => #Ziel);

           #nextStep := NOT #Befehl_ok;
       ELSE
           #nextStep := TRUE;
       END_IF;
       RETURN;
   END_IF;

   IF (#tmpQuelle = 20) OR (#tmpQuelle = 24) THEN
       //Kurz rechts
       #Vorzug := NOT #Positionen[25].Sperre AND NOT #Positionen[26].Sperre AND #Positionen[29].Sperre AND NOT #Positionen[30].Sperre;

       IF NOT #Positionen[26].Sperre AND NOT #Vorzug THEN
           "FC_FW_Auftrag_Befehl"(inQuelle := #tmpQuelle,
                                  inZiel := 26,
                                  Befehl_ok => #Befehl_ok,
                                  outQuelle => #Quelle,
                                  outZiel => #Ziel);

           #nextStep := NOT #Befehl_ok;
       ELSIF NOT #Positionen[30].Sperre THEN
           "FC_FW_Auftrag_Befehl"(inQuelle := #tmpQuelle,
                                  inZiel := 30,
                                  Befehl_ok => #Befehl_ok,
                                  outQuelle => #Quelle,
                                  outZiel => #Ziel);

           #nextStep := NOT #Befehl_ok;
       ELSE
           #nextStep := TRUE;
       END_IF;
       RETURN;
   END_IF;

   //?
   #nextStep := TRUE;
END_REGION
END_FUNCTION

FUNCTION "FC_FW_Auftrag_Suche" : Void   // FC180, LAD
{ S7_Optimized_Access := 'TRUE' }
// stored: AutoNumber false, SetENOAutomatically false
   VAR_INPUT
      Pos1 : Int;
      Pos2 : Int;
   END_VAR
   VAR_IN_OUT
      Positionen : Array[1..30] of "UDT_Auftrag_Pos";
      Quelle : Int;
      Oldest : Real;
   END_VAR
   VAR_TEMP
      Pos : Int;
   END_VAR
BEGIN

REGION Network 1 (SCL)
   FOR #Pos := #Pos1 TO #Pos2 DO
       IF #Positionen[#Pos].Abholbar AND NOT #Positionen[#Pos].CheckSperre THEN
           IF (#Quelle = 0) OR (#Positionen[#Pos].Oldest > #Oldest) THEN
               #Quelle := #Pos;
               #Oldest := #Positionen[#Pos].Oldest;
           END_IF;
       END_IF;
   END_FOR;
END_REGION
END_FUNCTION

FUNCTION "FC_KorrPos" : Void   // FC216, STL
{ S7_Optimized_Access := 'FALSE' }
// stored: AutoNumber false
   VAR_INPUT
      TW_Nr : Int;   // Fahrwagennummer
      IstPos : Byte;   // Istposition aus Messbaustein
      ErrCount : Byte;   // Messwert ungültig bei <>0
      Laser_on : Bool;   // Messwert neu --> Korrektur
   END_VAR
   VAR_IN_OUT
      PosInc : DInt;   // IstPosition TW
   END_VAR
   VAR_TEMP
      IstPosInc : DInt;
      CheckPosInc : DInt;
      Korrektur : DInt;
      CheckPosKorr : DInt;
      s_max : Real;   // Abstand zwischen den Pos.
      s_ist : Real;   // Abstand zur Istposition
      KorrDiff : Real;   // Differenz beider Korrekturwerte
      CheckPos : Int;
      FW_DB : Int;
   END_VAR
BEGIN

NETWORK
TITLE = Initialisieren
//Korrekturrechnung deaktiviert
      AN    "DB_KorrPos".Berechnung_ein;
      O     "DB_ANLAGE".BA.Mess_on;
      BEC;

//erster Durchlauf ohne Korrektur
      L     #IstPos;
      L     0;
      ==I;
      BEC;

//Messsystem liefert gerade keinen Messwert
      L     #ErrCount;
      L     0;
      <>I;
      ON    #Laser_on;
      BEC;


NETWORK
TITLE = Inkremente holen Istposition
      L     #IstPos;
      L     "DB_POS".LENG;
      *D;
      L     "DB_POS".Offset;
      +D;
      SLD   3;
      LAR1;
      OPN   "DB_POS";
      L     DBD [AR1, P#22.0];  //"DB_POS".POS[0].IncPos
      T     #IstPosInc;

      L     #TW_Nr;
      +     -1;
      L     "DB_KorrPos".Leng;
      *D;
      L     "DB_KorrPos".Offset;
      +D;
      SLD   3;
      LAR1;  //Adresse Start TWx
      OPN   "DB_KorrPos";
      L     #IstPos;
      +     -1;
      L     2;
      *D;
      SLD   3;
      +AR1;  //Adresse Posy zu TWx
      L     DBW [AR1, P#0.0];  //"DB_KorrPos".TW1[1].Pos[1]
      ITD;
      NEGD;  //Invertieren, weil positiver Offset negative Korrektur bedeutet
      T     #Korrektur;

      L     #PosInc;
      L     #IstPosInc;
      -D;
//höhere Pos testen
      JP    hPos;
//niedrigere Pos testen
      JM    nPos;
//genau mittig
      JU    Out;

//Höhere Position Testen
hPos: L     "DB_ANLAGE".config.ANZ_Pos;  //Es existiert keine größere Pos.
      L     #IstPos;
      <=I;
      JC    Out;
      +     1;
      T     #CheckPos;
      JU    Chk;

//Niedrigere Position Testen
nPos: L     1;  //Es existiert keine niedrigere Pos.
      L     #IstPos;
      >=I;
      JC    Out;
      +     -1;
      T     #CheckPos;
      JU    Chk;


NETWORK
TITLE = Checkposdaten holen
Chk:  L     #CheckPos;
      L     "DB_POS".LENG;
      *D;
      L     "DB_POS".Offset;
      +D;
      SLD   3;
      LAR1;
      OPN   "DB_POS";
      L     DBD [AR1, P#22.0];  //"DB_POS".POS[0].IncPos
      T     #CheckPosInc;

      L     #TW_Nr;
      +     -1;
      L     "DB_KorrPos".Leng;
      *D;
      L     "DB_KorrPos".Offset;
      +D;
      SLD   3;
      LAR1;  //Adresse Start TWx
      OPN   "DB_KorrPos";
      L     #CheckPos;
      +     -1;
      L     2;
      *D;
      SLD   3;
      +AR1;  //Adresse Posy zu TWx
      L     DBW [AR1, P#0.0];  //"DB_KorrPos".TW1[1].Pos[1]
      ITD;
      NEGD;  //Invertieren, weil positiver Offset negative Korrektur bedeutet
      T     #CheckPosKorr;


NETWORK
TITLE = Korrektur berechnen
      L     #IstPosInc;
      L     #Korrektur;
      -D;
      T     #IstPosInc;

      L     #CheckPosInc;
      L     #CheckPosKorr;
      -D;
      T     #CheckPosInc;

      L     #IstPosInc;
      L     #CheckPosInc;
      -D;
      DTR;
      ABS;
      T     #s_max;
      L     0.0;  //Div durch Null (beide Pos gleiches Inc)
      ==R;
      JC    Out;

      L     #IstPosInc;
      L     #PosInc;
      -D;
      DTR;
      ABS;
      T     #s_ist;

      L     #CheckPosKorr;
      L     #Korrektur;
      -D;
      DTR;
      T     #KorrDiff;

      L     #s_ist;
      L     #s_max;
      /R;
      L     #KorrDiff;
      *R;
      RND;
      L     #Korrektur;
      +D;
      T     #Korrektur;


NETWORK
TITLE = Ausgabe
Out:  L     #Korrektur;
      L     #PosInc;
      +D;
      T     #PosInc;

END_FUNCTION

FUNCTION "FC_Takt_periodisch" : Void   // FC26, STL
{ S7_Optimized_Access := 'FALSE' }
// stored: AutoNumber false
   VAR_INPUT
      Freigabe : Bool;   // Taktung einschalten
      Timer_Nr : Timer;   // Timer für Takt
      Zeit_ein : S5Time;   // Einschaltzeit
      Zeit_aus : S5Time;   // Pausenzeit
   END_VAR
   VAR_OUTPUT
      on : Bool;   // Ausgang getaktet
   END_VAR
BEGIN

NETWORK
TITLE = Ausgang getaktet
      AN    #Freigabe;
      L     #Zeit_aus;
      SF    #Timer_Nr;

      A     #Freigabe;
      L     #Zeit_ein;
      SD    #Timer_Nr;

      AN    #Timer_Nr;
      A     #Freigabe;
      =     #on;

END_FUNCTION

FUNCTION "AZ_on_off" : Void
{ S7_Optimized_Access := 'TRUE' }
VERSION : 0.1
   VAR_INPUT 
      Time_to_on : Int;   // Zeitpunkt der Einschaltung relativ zu AZ-Beginn (min)
      Time_to_off : Int;   // Zeitpunkt der Ausschaltung relativ zu AZ-Ende (min)
   END_VAR

   VAR_OUTPUT 
      on : Bool;
   END_VAR


BEGIN
	//-----------------------------------------------------
	//Ist gerade Arbeitszeit?
	//-----------------------------------------------------
	#on := "Uhrzeit".AZ_aktiv;
	
	IF "Uhrzeit".AZ_aktiv = true THEN
	    //-----------------------------------------------------
	    //Behandlung während Arbeitszeit
	    //-----------------------------------------------------
	    IF #Time_to_off < 0 AND ((#Time_to_off * -1) >= "Uhrzeit".Time_to_off) THEN
	        #on := FALSE;
	    END_IF;
	    
	    IF #Time_to_on >= 0 AND (#Time_to_on > ("Uhrzeit".Time_to_on * -1)) THEN
	        #on := FALSE;
	    END_IF;
	    
	ELSE
	    //-----------------------------------------------------
	    //Behandlung außerhalb Arbeitszeit
	    //-----------------------------------------------------
	    IF #Time_to_on < 0 AND ((#Time_to_on * -1) >= "Uhrzeit".Time_to_on) THEN
	        #on := TRUE;
	    END_IF;
	    
	    IF #Time_to_off >= 0 AND (#Time_to_off > ("Uhrzeit".Time_to_off * -1)) THEN
	        #on := TRUE;
	    END_IF;
	    
	END_IF;
	
END_FUNCTION

FUNCTION "Analogausgabe" : Void
{ S7_Optimized_Access := 'TRUE' }
VERSION : 0.1
   VAR_INPUT 
      Input_Value : Real;   // zu wandelnde Größe
      X_MIN : Real;
      X_MAX : Real;
      Y_UGR : Real;
      Y_OGR : Real;
   END_VAR

   VAR_OUTPUT 
      Output_Value : Int;
   END_VAR

   VAR_TEMP 
      Range : Real;
   END_VAR


BEGIN
	#Range := #X_MAX - #X_MIN;
	IF #Range = 0.0 THEN
	    #Output_Value := 0;
	ELSE
	    #Output_Value := UINT_TO_INT(ROUND_UINT(((#Input_Value - #X_MIN)* #Y_OGR / #Range ) + ((#X_MAX - #Input_Value) * #Y_UGR / #Range )));
	END_IF;
	 
END_FUNCTION

FUNCTION "Niv_Visu" : Void
{ S7_Optimized_Access := 'TRUE' }
VERSION : 0.1
   VAR_INPUT 
      Niv_1 : Bool;   // 1 == Niveau erreicht
      Niv_2 : Bool;   // 1 == Niveau erreicht
      Niv_3 : Bool;   // 1 == Niveau erreicht
      Niv_4 : Bool;   // 1 == Niveau erreicht
      Niv_5 : Bool;   // 1 == Niveau erreicht
      Niv_6 : Bool;   // 1 == Niveau erreicht
      Wert_1 : USInt;   // [%]
      Wert_2 : USInt;   // [%]
      Wert_3 : USInt;   // [%]
      Wert_4 : USInt;   // [%]
      Wert_5 : USInt;   // [%]
      Wert_6 : USInt;   // [%]
   END_VAR

   VAR_OUTPUT 
      Niveau : USInt;   // [%]
      Niv_Err : Bool;   // ein höheres Niveau ist an obwohl ein niedrigeres nicht an ist
   END_VAR


BEGIN
	//Analogwert - Prozentanzeige Visu
	IF #Niv_6 AND #Niv_5 AND #Niv_4 AND #Niv_3 AND #Niv_2 AND #Niv_1 THEN
	    #Niveau := #Wert_6;
	ELSIF NOT #Niv_6 AND #Niv_5 AND #Niv_4 AND #Niv_3 AND #Niv_2 AND #Niv_1 THEN
	    #Niveau := #Wert_5;
	ELSIF NOT #Niv_6 AND NOT #Niv_5 AND #Niv_4 AND #Niv_3 AND #Niv_2 AND #Niv_1 THEN
	    #Niveau := #Wert_4;
	ELSIF NOT #Niv_6 AND NOT #Niv_5 AND NOT #Niv_4 AND #Niv_3 AND #Niv_2 AND #Niv_1 THEN
	    #Niveau := #Wert_3;
	ELSIF NOT #Niv_6 AND NOT #Niv_5 AND NOT #Niv_4 AND NOT #Niv_3 AND #Niv_2 AND #Niv_1 THEN
	    #Niveau := #Wert_2;
	ELSIF NOT #Niv_6 AND NOT #Niv_5 AND NOT #Niv_4 AND NOT #Niv_3 AND NOT #Niv_2 AND #Niv_1 THEN
	    #Niveau := #Wert_1;
	ELSIF NOT #Niv_6 AND NOT #Niv_5 AND NOT #Niv_4 AND NOT #Niv_3 AND NOT #Niv_2 AND NOT #Niv_1 THEN
	    #Niveau := 0;
	ELSE
	    #Niveau := 150; //Fehler Niveau
	END_IF;
	
	//Plausibilitätsprüfung
	#Niv_Err := (#Niv_6 AND (NOT #Niv_5 OR NOT #Niv_4 OR NOT #Niv_3 OR NOT #Niv_2 OR NOT #Niv_1)) OR
	(#Niv_5 AND (NOT #Niv_4 OR NOT #Niv_3 OR NOT #Niv_2 OR NOT #Niv_1)) OR
	(#Niv_4 AND (NOT #Niv_3 OR NOT #Niv_2 OR NOT #Niv_1)) OR
	(#Niv_3 AND (NOT #Niv_2 OR NOT #Niv_1)) OR
	(#Niv_2 AND (NOT #Niv_1));
	
END_FUNCTION

FUNCTION "Status_E0A" : Void
{ S7_Optimized_Access := 'TRUE' }
VERSION : 0.1
   VAR_INPUT 
      Hand : Bool;
      Auto : Bool;
      SonderModus_PumpeSpuelen : Bool;
      Stoerung : Bool;   // 1 bei Fehler
      Ausgang : Bool;
   END_VAR

   VAR_OUTPUT 
      StatusByte : USInt;
   END_VAR

   VAR CONSTANT 
      Aus : USInt;
      Hand_EIN : USInt := 1;
      Hand_AUS : USInt := 2;
      Auto_EIN : USInt := 3;
      Auto_AUS : USInt := 4;
      Fehler : USInt := 5;
      Spuelen_aktiv : USInt := 10;
   END_VAR


BEGIN
	//Status für Visu
	IF (#Hand OR #Auto) AND #Stoerung THEN
	    #StatusByte := #Fehler;
	ELSIF #Auto AND NOT #Ausgang THEN
	    #StatusByte := #Auto_AUS;
	ELSIF #Ausgang AND #Auto THEN
	    #StatusByte := #Auto_EIN;
	ELSIF #Hand AND NOT #Ausgang AND #SonderModus_PumpeSpuelen THEN
	    #StatusByte := #Spuelen_aktiv;
	ELSIF #Hand AND NOT #Ausgang THEN
	    #StatusByte := #Hand_AUS;
	ELSIF #Hand AND #Ausgang THEN
	    #StatusByte := #Hand_EIN;
	ELSE
	    #StatusByte := #Aus;
	END_IF;
	
END_FUNCTION

